C08918=1012.059,211.488,-136.329,-51.249,85.122,-51.521
C08919=1012.057,211.246,-136.302,-51.186,85.113,-51.456
C08920=1012.055,211.003,-136.276,-51.123,85.104,-51.390
C08921=1012.053,210.760,-136.249,-51.059,85.095,-51.325
C08922=1012.051,210.518,-136.223,-50.990,85.086,-51.253
C08923=1012.049,210.275,-136.196,-50.928,85.077,-51.188
C08924=1012.046,210.033,-136.169,-50.865,85.068,-51.124
C08925=1012.044,209.791,-136.143,-50.803,85.060,-51.060
C08926=1012.042,209.548,-136.116,-50.748,85.051,-51.003
C08927=1012.040,209.306,-136.090,-50.679,85.041,-50.932
C08928=1012.037,209.063,-136.063,-50.618,85.032,-50.869
C08929=1012.036,208.821,-136.037,-50.557,85.024,-50.805
C08930=1012.034,208.578,-136.010,-50.495,85.014,-50.742
C08931=1012.032,208.336,-135.984,-50.441,85.007,-50.686
C08932=1012.030,208.093,-135.958,-50.374,84.997,-50.617
C08933=1012.027,207.851,-135.931,-50.314,84.988,-50.555
C08934=1012.025,207.608,-135.905,-50.254,84.979,-50.492
C08935=1012.023,207.365,-135.878,-50.194,84.970,-50.430
C08936=1012.021,207.122,-135.852,-50.134,84.961,-50.369
C08937=1012.020,206.880,-135.826,-50.074,84.951,-50.307
C08938=1012.018,206.636,-135.799,-50.015,84.943,-50.246
C08939=1012.016,206.393,-135.773,-49.956,84.934,-50.185
C08940=1012.014,206.150,-135.746,-49.897,84.924,-50.124
C08941=1012.011,205.906,-135.720,-49.838,84.915,-50.064
C08942=1012.010,205.663,-135.693,-49.780,84.907,-50.003
C08943=1012.008,205.419,-135.667,-49.716,84.897,-49.936
C08944=1012.005,205.175,-135.640,-49.658,84.888,-49.876
C08945=1012.004,204.930,-135.613,-49.600,84.878,-49.817
C08946=1012.002,204.687,-135.587,-49.542,84.870,-49.757
C08947=1011.999,204.443,-135.561,-49.485,84.860,-49.698
C08948=1011.998,204.198,-135.534,-49.422,84.851,-49.632
C08949=1011.996,203.954,-135.508,-49.365,84.841,-49.573
C08950=1011.994,203.710,-135.481,-49.308,84.833,-49.514
C08951=1011.992,203.464,-135.454,-49.251,84.823,-49.456
C08952=1011.987,202.215,-135.317,-47.331,85.025,-47.026
C08953=1011.988,201.996,-135.294,-47.276,85.015,-46.969
C08954=1011.988,201.790,-135.271,-47.227,85.007,-46.919
C08955=1011.988,201.373,-135.226,-47.131,84.989,-46.820
C08956=1011.989,201.157,-135.203,-47.083,84.981,-46.770
C08957=1011.989,200.933,-135.179,-47.029,84.971,-46.714
C08958=1011.989,200.695,-135.153,-46.976,84.962,-46.659
C08959=1011.989,200.439,-135.126,-46.922,84.951,-46.605
C08960=1011.990,200.186,-135.099,-46.863,84.940,-46.544
C08961=1011.989,199.944,-135.073,-46.811,84.930,-46.490
C08962=1011.990,199.712,-135.048,-46.758,84.921,-46.435
C08963=1011.990,199.483,-135.023,-46.705,84.911,-46.381
C08964=1011.990,199.241,-134.997,-46.653,84.902,-46.327
C08965=1011.991,198.850,-134.954,-46.566,84.885,-46.238
C08966=1011.991,198.458,-134.913,-46.486,84.869,-46.156
C08967=1011.992,198.212,-134.886,-46.429,84.859,-46.096
C08968=1011.992,197.976,-134.861,-46.378,84.848,-46.044
C08969=1011.992,197.740,-134.836,-46.327,84.838,-45.991
C08970=1011.992,197.504,-134.810,-46.276,84.829,-45.939
C08971=1011.993,197.268,-134.785,-46.226,84.818,-45.887
C08972=1011.993,197.032,-134.759,-46.175,84.808,-45.835
C08973=1011.993,196.796,-134.734,-46.125,84.799,-45.783
C08974=1011.993,196.560,-134.709,-46.075,84.789,-45.731
C08975=1011.994,196.324,-134.684,-46.031,84.780,-45.686
C08976=1011.994,196.088,-134.658,-45.981,84.770,-45.635
C08977=1011.995,195.852,-134.633,-45.932,84.761,-45.583
C08978=1011.995,195.616,-134.609,-45.883,84.750,-45.533
C08979=1011.995,195.380,-134.583,-45.834,84.740,-45.483
C08980=1011.996,195.144,-134.558,-45.785,84.731,-45.432
C08981=1011.996,194.908,-134.532,-45.742,84.721,-45.388
C08982=1011.996,194.673,-134.507,-45.693,84.711,-45.339
C08983=1011.997,194.437,-134.482,-45.645,84.701,-45.288
C08984=1011.997,194.201,-134.456,-45.602,84.692,-45.245
C08985=1011.998,193.965,-134.431,-45.554,84.682,-45.195
C08986=1011.997,193.729,-134.406,-45.512,84.673,-45.151
C08987=1011.998,193.492,-134.381,-45.464,84.663,-45.102
C08988=1011.999,193.257,-134.356,-45.417,84.653,-45.053
C08989=1011.999,193.021,-134.330,-45.370,84.643,-45.005
C08990=1011.999,192.785,-134.306,-45.323,84.633,-44.956
C08991=1011.999,192.549,-134.280,-45.281,84.624,-44.913
C08992=1012.000,192.313,-134.255,-45.235,84.614,-44.865
C08993=1012.000,192.077,-134.229,-45.188,84.604,-44.817
C08994=1012.000,191.841,-134.205,-45.147,84.595,-44.774
C08995=1012.001,191.605,-134.180,-45.106,84.586,-44.732
C08996=1012.001,191.369,-134.154,-45.060,84.576,-44.685
C08997=1012.002,191.133,-134.129,-45.019,84.567,-44.643
C08998=1012.002,190.898,-134.104,-44.974,84.556,-44.597
C08999=1012.002,190.662,-134.079,-44.928,84.546,-44.549
C09000=1012.003,190.425,-134.054,-44.883,84.537,-44.502
C09001=1012.004,190.189,-134.028,-44.838,84.527,-44.455
C09002=1012.003,189.954,-134.004,-44.798,84.517,-44.415
C09003=1012.004,189.718,-133.978,-44.759,84.507,-44.375
C09004=1012.004,189.482,-133.953,-44.714,84.498,-44.328
C09005=1012.005,189.245,-133.928,-44.674,84.488,-44.288
C09006=1012.006,189.010,-133.903,-44.635,84.480,-44.246
C09007=1012.006,188.774,-133.878,-44.591,84.469,-44.201
C09008=1012.006,188.538,-133.853,-44.547,84.459,-44.155
C09009=1012.007,188.302,-133.828,-44.508,84.450,-44.115
C09010=1012.007,188.066,-133.803,-44.464,84.439,-44.071
C09011=1012.007,187.830,-133.777,-44.421,84.430,-44.026
C09012=1012.008,187.595,-133.753,-44.382,84.420,-43.986
C09013=1012.008,187.359,-133.728,-44.344,84.411,-43.947
C09014=1012.009,187.123,-133.703,-44.306,84.402,-43.907
C09015=1012.010,186.887,-133.677,-44.263,84.392,-43.863
C09016=1012.009,186.651,-133.652,-44.225,84.383,-43.824
C09017=1012.011,186.415,-133.628,-44.187,84.373,-43.785
C09018=1012.011,186.179,-133.603,-44.145,84.363,-43.740
C09019=1012.011,185.943,-133.578,-44.103,84.353,-43.698
C09020=1012.011,185.707,-133.552,-44.065,84.343,-43.659
C09021=1012.013,185.472,-133.528,-44.023,84.334,-43.615
C09022=1012.012,185.236,-133.503,-43.986,84.324,-43.577
C09023=1012.013,185.000,-133.478,-43.949,84.315,-43.539
C09024=1012.014,184.763,-133.453,-43.912,84.306,-43.501
C09025=1012.014,184.528,-133.428,-43.876,84.296,-43.464
C09026=1012.015,184.292,-133.403,-43.839,84.287,-43.426
C09027=1012.015,184.057,-133.377,-43.798,84.277,-43.383
C09028=1012.015,183.820,-133.353,-43.756,84.267,-43.340
C09029=1012.016,183.585,-133.328,-43.721,84.257,-43.304
C09030=1012.017,183.349,-133.303,-43.685,84.248,-43.267
C09031=1012.017,183.113,-133.279,-43.644,84.238,-43.224
C09032=1012.018,182.877,-133.254,-43.608,84.228,-43.188
C09033=1012.018,182.642,-133.228,-43.573,84.219,-43.151
C09034=1012.018,182.405,-133.204,-43.537,84.210,-43.114
C09035=1012.019,182.170,-133.179,-43.502,84.200,-43.078
C09036=1012.020,181.934,-133.153,-43.466,84.191,-43.041
C09037=1012.020,181.698,-133.129,-43.431,84.182,-43.005
C09038=1012.021,181.462,-133.104,-43.391,84.172,-42.963
C09039=1012.021,181.227,-133.079,-43.356,84.162,-42.927
C09040=1012.021,180.990,-133.055,-43.317,84.152,-42.888
C09041=1012.023,180.755,-133.029,-43.283,84.142,-42.852
C09042=1012.023,180.519,-133.005,-43.248,84.133,-42.816
C09043=1012.024,180.283,-132.980,-43.214,84.123,-42.781
C09044=1012.024,180.047,-132.955,-43.179,84.114,-42.745
C09045=1012.024,179.811,-132.931,-43.149,84.106,-42.714
C09046=1012.025,179.576,-132.905,-43.115,84.097,-42.679
C09047=1012.026,179.340,-132.880,-43.077,84.086,-42.640
C09048=1012.026,179.104,-132.856,-43.043,84.077,-42.605
C09049=1012.027,178.868,-132.831,-43.009,84.067,-42.570
C09050=1012.027,178.632,-132.807,-42.971,84.057,-42.530
C09051=1012.028,178.397,-132.782,-42.937,84.048,-42.495
C09052=1012.028,178.161,-132.756,-42.904,84.038,-42.461
C09053=1012.029,177.925,-132.732,-42.875,84.030,-42.432
C09054=1012.030,177.689,-132.707,-42.842,84.020,-42.397
C09055=1012.030,177.454,-132.683,-42.809,84.011,-42.363
C09056=1012.031,177.218,-132.658,-42.776,84.001,-42.329
C09057=1012.032,176.982,-132.633,-42.743,83.992,-42.295
C09058=1012.032,176.746,-132.608,-42.705,83.982,-42.256
C09059=1012.033,176.511,-132.583,-42.673,83.973,-42.222
C09060=1012.033,176.275,-132.559,-42.641,83.962,-42.190
C09061=1012.034,176.040,-132.534,-42.608,83.953,-42.157
C09062=1012.034,175.803,-132.510,-42.576,83.943,-42.123
C09063=1012.035,175.568,-132.485,-42.547,83.936,-42.094
C09064=1012.036,175.331,-132.460,-42.515,83.926,-42.060
C09065=1012.036,175.096,-132.436,-42.483,83.917,-42.027
C09066=1012.037,174.860,-132.410,-42.451,83.907,-41.994
C09067=1012.037,174.625,-132.386,-42.419,83.898,-41.961
C09068=1012.038,174.389,-132.361,-42.388,83.888,-41.930
C09069=1012.038,174.153,-132.337,-42.357,83.878,-41.897
C09070=1012.039,173.917,-132.312,-42.325,83.869,-41.865
C09071=1012.040,173.682,-132.288,-42.294,83.859,-41.832
C09072=1012.040,173.446,-132.262,-42.267,83.850,-41.805
C09073=1012.041,173.210,-132.239,-42.235,83.842,-41.771
C09074=1012.042,172.975,-132.214,-42.204,83.832,-41.739
C09075=1012.043,172.738,-132.189,-42.177,83.824,-41.712
C09076=1012.043,172.504,-132.164,-42.146,83.814,-41.680
C09077=1012.044,172.267,-132.140,-42.115,83.805,-41.648
C09078=1012.044,172.032,-132.115,-42.085,83.794,-41.618
C09079=1012.045,171.796,-132.091,-42.054,83.785,-41.586
C09080=1012.045,171.560,-132.066,-42.024,83.775,-41.554
C09081=1012.047,171.325,-132.041,-41.993,83.766,-41.523
C09082=1012.047,171.090,-132.017,-41.966,83.758,-41.495
C09083=1012.047,170.854,-131.991,-41.936,83.749,-41.463
C09084=1012.048,170.618,-131.968,-41.910,83.740,-41.437
C09085=1012.049,170.383,-131.943,-41.880,83.730,-41.406
C09086=1012.049,170.147,-131.918,-41.850,83.721,-41.375
C09087=1012.050,169.911,-131.894,-41.820,83.711,-41.344
C09088=1012.051,169.676,-131.870,-41.790,83.702,-41.313
C09089=1012.051,169.439,-131.845,-41.765,83.693,-41.287
C09090=1012.052,169.204,-131.820,-41.735,83.683,-41.256
C09091=1012.053,168.969,-131.797,-41.705,83.674,-41.226
C09092=1012.053,168.733,-131.771,-41.680,83.665,-41.200
C09093=1012.054,168.497,-131.747,-41.651,83.656,-41.170
C09094=1012.055,168.262,-131.722,-41.625,83.648,-41.143
C09095=1012.055,168.026,-131.698,-41.600,83.639,-41.117
C09096=1012.056,167.790,-131.673,-41.571,83.629,-41.087
C09097=1012.057,167.555,-131.649,-41.542,83.619,-41.059
C09098=1012.058,167.319,-131.624,-41.513,83.609,-41.029
C09099=1012.058,167.083,-131.600,-41.485,83.600,-40.999
C09100=1012.058,166.848,-131.576,-41.460,83.591,-40.974
C09101=1012.059,166.612,-131.551,-41.430,83.582,-40.942
C09102=1012.060,166.377,-131.527,-41.406,83.573,-40.917
C09103=1012.061,166.142,-131.502,-41.381,83.565,-40.893
C09104=1012.061,165.906,-131.477,-41.353,83.555,-40.863
C09105=1012.062,165.670,-131.453,-41.328,83.547,-40.837
C09106=1012.063,165.434,-131.429,-41.299,83.538,-40.808
C09107=1012.063,165.200,-131.405,-41.275,83.529,-40.783
C09108=1012.064,164.896,-131.373,-41.240,83.517,-40.746
C09109=1012.065,164.578,-131.340,-41.210,83.505,-40.716
C09110=1012.066,164.304,-131.312,-41.179,83.494,-40.684
C09111=1012.067,163.969,-131.277,-41.141,83.481,-40.645
C09112=1012.068,163.749,-131.254,-41.116,83.473,-40.619
C09113=1012.068,163.511,-131.230,-41.092,83.464,-40.595
C09114=1012.069,163.247,-131.202,-41.062,83.453,-40.563
C09115=1012.071,162.954,-131.172,-41.031,83.442,-40.532
C09116=1012.070,162.646,-131.140,-41.001,83.431,-40.501
C09117=1012.072,162.355,-131.110,-40.966,83.419,-40.465
C09118=1012.073,162.048,-131.079,-40.937,83.407,-40.436
C09119=1012.073,161.745,-131.047,-40.903,83.395,-40.400
C09120=1012.075,161.453,-131.017,-40.873,83.384,-40.369
C09121=1012.076,161.175,-130.988,-40.843,83.373,-40.339
C09122=1012.076,160.912,-130.961,-40.816,83.363,-40.311
C09123=1012.077,160.663,-130.935,-40.791,83.353,-40.285
C09124=1012.078,160.422,-130.911,-40.764,83.343,-40.257
C09125=1012.079,160.188,-130.887,-40.741,83.334,-40.234
C09126=1012.080,159.956,-130.865,-40.625,83.289,-40.116
C09127=1012.080,159.723,-130.845,-40.392,83.195,-39.879
C09128=1012.082,159.489,-130.825,-40.163,83.099,-39.646
C09129=1012.083,159.253,-130.805,-39.936,83.004,-39.413
C09130=1012.084,159.017,-130.786,-39.720,82.908,-39.193
C09131=1012.085,158.781,-130.765,-39.510,82.812,-38.979
C09132=1012.086,158.546,-130.745,-39.305,82.716,-38.770
C09133=1012.087,158.311,-130.725,-39.107,82.620,-38.568
C09134=1012.089,158.074,-130.705,-38.914,82.523,-38.371
C09135=1012.090,157.837,-130.685,-38.721,82.427,-38.174
C09136=1012.092,157.599,-130.665,-38.539,82.330,-37.988
C09137=1012.092,157.360,-130.644,-38.358,82.233,-37.803
C09138=1012.093,157.121,-130.624,-38.181,82.135,-37.623
C09139=1012.095,156.882,-130.604,-38.010,82.037,-37.448
C09140=1012.096,156.643,-130.584,-37.842,81.939,-37.277
C09141=1012.097,156.403,-130.563,-37.680,81.841,-37.110
C09142=1012.099,156.163,-130.543,-37.524,81.743,-36.952
C09143=1012.100,155.924,-130.523,-37.368,81.646,-36.792
C09144=1012.101,155.685,-130.503,-37.217,81.548,-36.638
C09145=1012.102,155.446,-130.483,-37.071,81.451,-36.489
C09146=1012.104,155.205,-130.463,-36.927,81.352,-36.342
C09147=1012.105,154.965,-130.442,-36.787,81.253,-36.199
C09148=1012.106,154.725,-130.422,-36.652,81.156,-36.061
C09149=1012.108,154.484,-130.402,-36.518,81.057,-35.925
C09150=1012.109,154.243,-130.381,-36.387,80.959,-35.790
C09151=1012.110,154.002,-130.361,-36.262,80.860,-35.663
C09152=1012.112,153.761,-130.340,-36.136,80.762,-35.534
C09153=1012.113,153.520,-130.320,-36.013,80.664,-35.408
C09154=1012.115,153.277,-130.299,-35.897,80.565,-35.290
C09155=1012.116,153.037,-130.279,-35.780,80.466,-35.170
C09156=1012.118,152.794,-130.259,-35.665,80.368,-35.053
C09157=1012.119,152.553,-130.238,-35.557,80.269,-34.943
C09158=1012.121,152.309,-130.217,-35.447,80.170,-34.831
C09159=1012.122,152.060,-130.196,-35.338,80.068,-34.720
C09160=1012.124,151.805,-130.176,-35.230,79.964,-34.610
C09161=1012.125,151.548,-130.154,-35.122,79.859,-34.500
C09162=1012.126,151.284,-130.131,-35.013,79.751,-34.389
C09163=1012.128,150.992,-130.107,-34.898,79.633,-34.272
C09164=1012.130,150.706,-130.082,-34.786,79.517,-34.158
C09165=1012.132,150.413,-130.057,-34.676,79.397,-34.046
C09166=1012.134,150.117,-130.032,-34.568,79.277,-33.937
C09167=1012.136,149.816,-130.007,-34.461,79.155,-33.828
C09168=1012.137,149.517,-129.981,-34.355,79.033,-33.721
C09169=1012.139,149.217,-129.956,-34.252,78.911,-33.615
C09170=1012.141,148.921,-129.931,-34.154,78.791,-33.517
C09171=1012.143,148.630,-129.907,-34.060,78.672,-33.422
C09172=1012.145,148.344,-129.883,-33.969,78.557,-33.329
C09173=1012.147,148.066,-129.859,-33.883,78.443,-33.242
C09174=1012.149,147.796,-129.837,-33.801,78.334,-33.160
C09175=1012.150,147.535,-129.814,-33.724,78.228,-33.082
C09176=1012.152,147.280,-129.793,-33.650,78.125,-33.007
C09177=1012.153,147.032,-129.772,-33.581,78.024,-32.938
C09178=1012.154,146.788,-129.751,-33.512,77.925,-32.869
C09179=1012.156,146.546,-129.731,-33.445,77.828,-32.801
C09180=1012.158,146.303,-129.710,-33.381,77.730,-32.737
C09181=1012.159,146.061,-129.690,-33.317,77.632,-32.674
C09182=1012.162,145.819,-129.670,-33.254,77.534,-32.610
C09183=1012.163,145.577,-129.649,-33.193,77.436,-32.549
C09184=1012.164,145.335,-129.629,-33.132,77.338,-32.488
C09185=1012.166,145.093,-129.608,-33.073,77.242,-32.430
C09186=1012.168,144.852,-129.588,-33.014,77.144,-32.371
C09187=1012.170,144.611,-129.568,-32.959,77.046,-32.317
C09188=1012.171,144.369,-129.547,-32.903,76.949,-32.262
C09189=1012.172,144.128,-129.527,-32.846,76.852,-32.204
C09190=1012.174,143.887,-129.506,-32.793,76.755,-32.151
C09191=1012.176,143.647,-129.486,-32.741,76.659,-32.101
C09192=1012.178,143.406,-129.466,-32.689,76.562,-32.049
C09193=1012.179,143.166,-129.446,-32.638,76.465,-31.999
C09194=1012.181,142.925,-129.425,-32.588,76.370,-31.950
C09195=1012.183,142.686,-129.404,-32.539,76.272,-31.902
C09196=1012.185,142.446,-129.385,-32.490,76.176,-31.855
C09197=1012.186,142.207,-129.365,-32.443,76.081,-31.808
C09198=1012.188,141.968,-129.344,-32.396,75.985,-31.763
C09199=1012.190,141.729,-129.324,-32.351,75.889,-31.718
C09200=1012.192,141.484,-129.304,-32.305,75.791,-31.675
C09201=1012.193,141.273,-129.286,-32.265,75.707,-31.635
C09202=1012.195,141.017,-129.264,-32.219,75.605,-31.591
C09203=1012.196,140.845,-129.249,-32.188,75.536,-31.561
C09204=1012.199,140.472,-129.219,-32.123,75.387,-31.499
C09205=1012.201,140.197,-129.195,-32.074,75.279,-31.452
C09206=1012.203,139.902,-129.170,-32.023,75.160,-31.403
C09207=1012.206,139.593,-129.144,-31.973,75.037,-31.355
C09208=1012.208,139.280,-129.118,-31.922,74.913,-31.307
C09209=1012.211,138.972,-129.092,-31.873,74.791,-31.261
C09210=1012.213,138.678,-129.067,-31.826,74.674,-31.216
C09211=1012.214,138.404,-129.044,-31.784,74.565,-31.177
C09212=1012.216,138.152,-129.022,-31.747,74.466,-31.143
C09213=1012.220,137.732,-128.987,-31.684,74.299,-31.084
C09214=1012.223,137.348,-128.955,-31.630,74.147,-31.034
C09215=1012.226,136.931,-128.919,-31.571,73.983,-30.980
C09216=1012.228,136.548,-128.887,-31.518,73.831,-30.932
C09217=1012.232,136.162,-128.854,-31.466,73.679,-30.883
C09218=1012.235,135.743,-128.819,-31.413,73.514,-30.837
C09219=1012.237,135.518,-128.801,-31.383,73.426,-30.810
C09220=1012.239,135.285,-128.781,-31.354,73.335,-30.784
C09221=1012.241,134.999,-128.756,-31.318,73.222,-30.752
C09222=1012.243,134.704,-128.731,-31.282,73.106,-30.720
C09223=1012.245,134.464,-128.711,-31.254,73.013,-30.696
C09224=1012.247,134.229,-128.691,-31.225,72.921,-30.670
C09225=1012.249,133.993,-128.672,-31.198,72.830,-30.647
C09226=1012.251,133.758,-128.652,-31.171,72.738,-30.623
C09227=1012.253,133.523,-128.632,-31.145,72.646,-30.602
C09228=1012.254,133.288,-128.612,-31.118,72.555,-30.578
C09229=1012.257,133.053,-128.592,-31.092,72.464,-30.556
C09230=1012.258,132.817,-128.573,-31.067,72.372,-30.535
C09231=1012.260,132.582,-128.553,-31.042,72.280,-30.513
C09232=1012.262,132.347,-128.533,-31.017,72.189,-30.493
C09233=1012.264,132.112,-128.513,-30.992,72.099,-30.472
C09234=1012.266,131.876,-128.493,-30.968,72.007,-30.452
C09235=1012.268,131.641,-128.473,-30.944,71.917,-30.432
C09236=1012.270,131.406,-128.453,-30.921,71.826,-30.414
C09237=1012.271,131.171,-128.433,-30.897,71.735,-30.393
C09238=1012.274,130.936,-128.413,-30.874,71.644,-30.376
C09239=1012.275,130.701,-128.393,-30.851,71.554,-30.358
C09240=1012.278,130.466,-128.373,-30.829,71.463,-30.340
C09241=1012.279,130.230,-128.353,-30.807,71.373,-30.322
C09242=1012.282,129.995,-128.333,-30.785,71.283,-30.306
C09243=1012.283,129.760,-128.314,-30.764,71.193,-30.289
C09244=1012.286,129.525,-128.294,-30.742,71.103,-30.272
C09245=1012.287,129.289,-128.274,-30.722,71.013,-30.257
C09246=1012.290,129.054,-128.254,-30.701,70.923,-30.242
C09247=1012.291,128.819,-128.234,-30.680,70.833,-30.226
C09248=1012.293,128.584,-128.214,-30.660,70.744,-30.210
C09249=1012.295,128.349,-128.195,-30.640,70.654,-30.196
C09250=1012.297,128.114,-128.175,-30.621,70.565,-30.182
C09251=1012.299,127.878,-128.155,-30.601,70.476,-30.167
C09252=1012.301,127.643,-128.135,-30.582,70.387,-30.153
C09253=1012.303,127.408,-128.115,-30.563,70.297,-30.140
C09254=1012.305,127.173,-128.095,-30.544,70.209,-30.127
C09255=1012.307,126.937,-128.075,-30.525,70.120,-30.113
C09256=1012.309,126.702,-128.056,-30.508,70.030,-30.103
C09257=1012.312,126.467,-128.036,-30.489,69.941,-30.089
C09258=1012.313,126.232,-128.016,-30.472,69.853,-30.078
C09259=1012.316,125.997,-127.996,-30.454,69.765,-30.066
C09260=1012.317,125.762,-127.975,-30.437,69.676,-30.055
C09261=1012.319,125.527,-127.956,-30.420,69.588,-30.044
C09262=1012.321,125.292,-127.935,-30.402,69.500,-30.031
C09263=1012.323,125.057,-127.916,-30.386,69.412,-30.021
C09264=1012.326,124.822,-127.896,-30.369,69.324,-30.011
C09265=1012.327,124.587,-127.877,-30.353,69.237,-30.000
C09266=1012.330,124.352,-127.857,-30.336,69.148,-29.991
C09267=1012.332,124.116,-127.836,-30.320,69.061,-29.981
C09268=1012.334,123.881,-127.817,-30.304,68.973,-29.971
C09269=1012.336,123.645,-127.797,-30.289,68.886,-29.962
C09270=1012.338,123.411,-127.777,-30.273,68.799,-29.953
C09271=1012.340,123.176,-127.757,-30.258,68.711,-29.945
C09272=1012.342,122.940,-127.737,-30.243,68.624,-29.937
C09273=1012.344,122.705,-127.718,-30.228,68.537,-29.928
C09274=1012.346,122.470,-127.697,-30.213,68.450,-29.920
C09275=1012.348,122.235,-127.678,-30.198,68.363,-29.911
C09276=1012.350,122.001,-127.657,-30.184,68.277,-29.905
C09277=1012.353,121.692,-127.631,-30.165,68.164,-29.895
C09278=1012.357,121.295,-127.598,-30.141,68.018,-29.883
C09279=1012.359,121.059,-127.577,-30.128,67.931,-29.877
C09280=1012.361,120.825,-127.558,-30.114,67.844,-29.870
C09281=1012.363,120.589,-127.538,-30.100,67.754,-29.864
C09282=1012.365,120.354,-127.518,-30.085,67.660,-29.856
C09283=1012.368,120.119,-127.499,-30.070,67.567,-29.850
C09284=1012.369,119.884,-127.480,-30.056,67.472,-29.845
C09285=1012.372,119.649,-127.460,-30.042,67.379,-29.839
C09286=1012.374,119.414,-127.441,-30.027,67.286,-29.832
C09287=1012.376,119.179,-127.420,-30.014,67.193,-29.827
C09288=1012.378,118.943,-127.402,-30.000,67.099,-29.822
C09289=1012.381,118.708,-127.382,-29.987,67.006,-29.817
C09290=1012.383,118.473,-127.362,-29.973,66.912,-29.811
C09291=1012.385,118.239,-127.342,-29.960,66.820,-29.807
C09292=1012.388,118.003,-127.323,-29.947,66.727,-29.803
C09293=1012.390,117.768,-127.304,-29.933,66.635,-29.797
C09294=1012.392,117.533,-127.284,-29.920,66.541,-29.793
C09295=1012.394,117.298,-127.264,-29.908,66.449,-29.791
C09296=1012.397,117.063,-127.244,-29.895,66.357,-29.786
C09297=1012.399,116.828,-127.226,-29.883,66.264,-29.783
C09298=1012.401,116.593,-127.206,-29.870,66.172,-29.780
C09299=1012.404,116.357,-127.185,-29.858,66.080,-29.778
C09300=1012.405,116.122,-127.166,-29.845,65.987,-29.774
C09301=1012.408,115.887,-127.147,-29.834,65.897,-29.772
C09302=1012.410,115.652,-127.127,-29.822,65.804,-29.770
C09303=1012.413,115.417,-127.108,-29.810,65.712,-29.767
C09304=1012.415,115.182,-127.088,-29.799,65.620,-29.765
C09305=1012.417,114.947,-127.068,-29.787,65.529,-29.764
C09306=1012.420,114.711,-127.049,-29.776,65.438,-29.761
C09307=1012.422,114.476,-127.029,-29.765,65.347,-29.760
C09308=1012.424,114.241,-127.009,-29.754,65.256,-29.760
C09309=1012.427,114.006,-126.989,-29.742,65.165,-29.756
C09310=1012.429,113.772,-126.970,-29.731,65.073,-29.756
C09311=1012.432,113.536,-126.951,-29.720,64.982,-29.755
C09312=1012.434,113.301,-126.932,-29.709,64.892,-29.754
C09313=1012.436,113.066,-126.911,-29.699,64.802,-29.755
C09314=1012.438,112.831,-126.891,-29.688,64.711,-29.753
C09315=1012.440,112.596,-126.872,-29.678,64.620,-29.754
C09316=1012.443,112.360,-126.853,-29.667,64.531,-29.754
C09317=1012.446,112.125,-126.833,-29.657,64.440,-29.755
C09318=1012.447,111.891,-126.813,-29.647,64.350,-29.754
C09319=1012.450,111.656,-126.794,-29.637,64.260,-29.755
C09320=1012.451,111.420,-126.774,-29.627,64.171,-29.755
C09321=1012.454,111.185,-126.755,-29.617,64.081,-29.756
C09322=1012.457,110.950,-126.735,-29.607,63.991,-29.757
C09323=1012.459,110.715,-126.715,-29.597,63.902,-29.758
C09324=1012.461,110.480,-126.695,-29.588,63.813,-29.760
C09325=1012.464,110.245,-126.675,-29.578,63.723,-29.761
C09326=1012.466,110.010,-126.657,-29.569,63.634,-29.763
C09327=1012.469,109.775,-126.637,-29.559,63.545,-29.763
C09328=1012.471,109.539,-126.617,-29.550,63.456,-29.766
C09329=1012.473,109.304,-126.597,-29.541,63.367,-29.769
C09330=1012.475,109.069,-126.577,-29.531,63.279,-29.770
C09331=1012.478,108.834,-126.557,-29.522,63.190,-29.773
C09332=1012.480,108.599,-126.539,-29.513,63.102,-29.775
C09333=1012.483,108.364,-126.519,-29.504,63.014,-29.777
C09334=1012.486,108.129,-126.499,-29.495,62.926,-29.781
C09335=1012.487,107.894,-126.479,-29.486,62.837,-29.783
C09336=1012.489,107.658,-126.459,-29.478,62.750,-29.786
C09337=1012.492,107.423,-126.440,-29.469,62.663,-29.789
C09338=1012.495,107.188,-126.420,-29.460,62.574,-29.792
C09339=1012.497,106.953,-126.401,-29.452,62.487,-29.795
C09340=1012.499,106.718,-126.381,-29.443,62.399,-29.799
C09341=1012.503,106.403,-126.354,-29.432,62.282,-29.805
C09342=1012.506,106.012,-126.322,-29.418,62.138,-29.811
C09343=1012.509,105.777,-126.302,-29.410,62.051,-29.814
C09344=1012.511,105.542,-126.283,-29.402,61.964,-29.819
C09345=1012.513,105.307,-126.263,-29.394,61.877,-29.823
C09346=1012.516,105.072,-126.243,-29.386,61.791,-29.827
C09347=1012.519,104.837,-126.223,-29.378,61.704,-29.832
C09348=1012.521,104.602,-126.204,-29.370,61.618,-29.836
C09349=1012.524,104.367,-126.184,-29.362,61.532,-29.841
C09350=1012.526,104.131,-126.164,-29.354,61.445,-29.846
C09351=1012.528,103.896,-126.144,-29.346,61.359,-29.851
C09352=1012.530,103.662,-126.125,-29.339,61.274,-29.856
C09353=1012.533,103.426,-126.105,-29.331,61.188,-29.861
C09354=1012.536,103.191,-126.085,-29.323,61.103,-29.866
C09355=1012.538,102.956,-126.065,-29.316,61.017,-29.872
C09356=1012.540,102.721,-126.046,-29.308,60.932,-29.878
C09357=1012.542,102.486,-126.026,-29.301,60.846,-29.883
C09358=1012.545,102.251,-126.006,-29.294,60.762,-29.890
C09359=1012.548,102.015,-125.987,-29.286,60.677,-29.894
C09360=1012.550,101.780,-125.967,-29.279,60.592,-29.901
C09361=1012.552,101.545,-125.947,-29.271,60.507,-29.905
C09362=1012.555,101.310,-125.927,-29.264,60.423,-29.913
C09363=1012.557,101.075,-125.907,-29.257,60.339,-29.919
C09364=1012.559,100.840,-125.888,-29.250,60.254,-29.925
C09365=1012.562,100.604,-125.869,-29.243,60.170,-29.931
C09366=1012.564,100.369,-125.849,-29.235,60.086,-29.937
C09367=1012.567,100.134,-125.829,-29.228,60.003,-29.944
C09368=1012.569,99.900,-125.809,-29.222,59.920,-29.951
C09369=1012.571,99.664,-125.789,-29.214,59.836,-29.957
C09370=1012.573,99.429,-125.769,-29.208,59.753,-29.965
C09371=1012.576,99.193,-125.750,-29.201,59.669,-29.971
C09372=1012.579,98.958,-125.730,-29.194,59.586,-29.979
C09373=1012.581,98.724,-125.711,-29.187,59.503,-29.987
C09374=1012.583,98.488,-125.690,-29.181,59.421,-29.993
C09375=1012.586,98.253,-125.670,-29.174,59.338,-30.001
C09376=1012.588,98.018,-125.650,-29.167,59.257,-30.008
C09377=1012.591,97.782,-125.631,-29.161,59.174,-30.016
C09378=1012.593,97.548,-125.612,-29.154,59.092,-30.024
C09379=1012.595,97.312,-125.591,-29.147,59.010,-30.030
C09380=1012.598,97.077,-125.572,-29.141,58.928,-30.040
C09381=1012.600,96.842,-125.552,-29.135,58.847,-30.047
C09382=1012.603,96.607,-125.532,-29.128,58.765,-30.055
C09383=1012.606,96.371,-125.512,-29.122,58.684,-30.063
C09384=1012.607,96.136,-125.493,-29.115,58.602,-30.071
C09385=1012.610,95.901,-125.473,-29.109,58.522,-30.080
C09386=1012.612,95.666,-125.453,-29.103,58.441,-30.087
C09387=1012.615,95.431,-125.433,-29.097,58.360,-30.096
C09388=1012.617,95.195,-125.413,-29.090,58.280,-30.105
C09389=1012.619,94.960,-125.394,-29.084,58.200,-30.112
C09390=1012.622,94.725,-125.374,-29.078,58.119,-30.122
C09391=1012.624,94.490,-125.354,-29.072,58.039,-30.130
C09392=1012.627,94.254,-125.334,-29.066,57.959,-30.139
C09393=1012.629,94.019,-125.314,-29.060,57.880,-30.148
C09394=1012.632,93.784,-125.294,-29.053,57.800,-30.156
C09395=1012.635,93.549,-125.275,-29.047,57.721,-30.165
C09396=1012.636,93.313,-125.255,-29.041,57.642,-30.174
C09397=1012.639,93.078,-125.235,-29.035,57.563,-30.183
C09398=1012.641,92.843,-125.215,-29.030,57.484,-30.193
C09399=1012.644,92.608,-125.195,-29.024,57.404,-30.202
C09400=1012.646,92.373,-125.175,-29.018,57.325,-30.211
C09401=1012.649,92.137,-125.156,-29.012,57.246,-30.221
C09402=1012.651,91.902,-125.136,-29.006,57.169,-30.229
C09403=1012.653,91.667,-125.116,-29.000,57.090,-30.240
C09404=1012.655,91.432,-125.096,-28.994,57.013,-30.249
C09405=1012.658,91.197,-125.076,-28.988,56.934,-30.259
C09406=1012.660,90.960,-125.056,-28.983,56.857,-30.268
C09407=1012.663,90.701,-125.034,-28.977,56.771,-30.280
C09408=1012.666,90.382,-125.008,-28.969,56.666,-30.292
C09409=1012.670,90.049,-124.979,-28.961,56.557,-30.306
C09410=1012.673,89.669,-124.947,-28.952,56.432,-30.323
C09411=1012.677,89.296,-124.916,-28.943,56.311,-30.340
C09412=1012.680,89.066,-124.896,-28.937,56.236,-30.350
C09413=1012.682,88.840,-124.877,-28.932,56.163,-30.359
C09414=1012.684,88.615,-124.858,-28.927,56.090,-30.369
C09415=1012.686,88.390,-124.839,-28.921,56.018,-30.379
C09416=1012.689,88.168,-124.820,-28.916,55.946,-30.388
C09417=1012.691,87.942,-124.802,-28.911,55.873,-30.398
C09418=1012.693,87.716,-124.782,-28.905,55.801,-30.409
C09419=1012.695,87.485,-124.763,-28.900,55.726,-30.420
C09420=1012.699,87.251,-124.743,-28.895,55.652,-30.431
C09421=1012.701,87.015,-124.723,-28.889,55.577,-30.441
C09422=1012.703,86.777,-124.702,-28.884,55.501,-30.451
C09423=1012.706,86.539,-124.683,-28.878,55.425,-30.462
C09424=1012.707,86.299,-124.662,-28.873,55.350,-30.473
C09425=1012.710,86.059,-124.642,-28.867,55.274,-30.485
C09426=1012.712,85.820,-124.621,-28.862,55.199,-30.495
C09427=1012.715,85.580,-124.601,-28.857,55.123,-30.507
C09428=1012.717,85.339,-124.581,-28.851,55.048,-30.518
C09429=1012.720,85.098,-124.561,-28.846,54.972,-30.530
C09430=1012.723,84.857,-124.541,-28.840,54.897,-30.541
C09431=1012.724,84.614,-124.520,-28.835,54.821,-30.553
C09432=1012.727,84.372,-124.500,-28.829,54.745,-30.564
C09433=1012.729,84.129,-124.478,-28.824,54.670,-30.575
C09434=1012.732,83.885,-124.458,-28.819,54.594,-30.588
C09435=1012.734,83.641,-124.437,-28.813,54.520,-30.599
C09436=1012.736,83.397,-124.416,-28.808,54.444,-30.612
C09437=1012.740,83.152,-124.396,-28.802,54.368,-30.623
C09438=1012.742,82.907,-124.375,-28.797,54.293,-30.634
C09439=1012.744,82.661,-124.354,-28.792,54.218,-30.648
C09440=1012.747,82.415,-124.333,-28.786,54.143,-30.659
C09441=1012.749,82.169,-124.312,-28.781,54.068,-30.671
C09442=1012.752,81.923,-124.292,-28.776,53.993,-30.685
C09443=1012.754,81.676,-124.271,-28.770,53.918,-30.696
C09444=1012.756,81.429,-124.250,-28.765,53.843,-30.708
C09445=1012.759,81.186,-124.230,-28.760,53.771,-30.720
C09446=1012.761,80.957,-124.210,-28.755,53.701,-30.733
C09447=1012.762,80.741,-124.191,-28.750,53.637,-30.743
C09448=1012.765,80.523,-124.173,-28.746,53.571,-30.755
C09449=1012.768,80.294,-124.154,-28.741,53.503,-30.767
C09450=1012.770,80.052,-124.133,-28.735,53.430,-30.779
C09451=1012.773,79.805,-124.112,-28.730,53.357,-30.791
C09452=1012.775,79.560,-124.092,-28.725,53.285,-30.804
C09453=1012.777,79.319,-124.071,-28.720,53.214,-30.816
C09454=1012.779,79.079,-124.050,-28.715,53.143,-30.828
C09455=1012.781,78.842,-124.030,-28.710,53.073,-30.841
C09456=1012.784,78.607,-124.010,-28.705,53.003,-30.854
C09457=1012.786,78.375,-123.990,-28.700,52.937,-30.865
C09458=1012.789,78.144,-123.971,-28.695,52.869,-30.877
C09459=1012.791,77.916,-123.952,-28.691,52.803,-30.889
C09460=1012.793,77.689,-123.932,-28.686,52.736,-30.901
C09461=1012.795,77.461,-123.913,-28.681,52.670,-30.913
C09462=1012.797,77.234,-123.893,-28.676,52.604,-30.925
C09463=1012.799,77.005,-123.875,-28.671,52.538,-30.937
C09464=1012.802,76.775,-123.855,-28.667,52.471,-30.950
C09465=1012.804,76.542,-123.835,-28.662,52.405,-30.962
C09466=1012.807,76.307,-123.816,-28.657,52.337,-30.975
C09467=1012.808,76.069,-123.795,-28.652,52.269,-30.988
C09468=1012.811,75.827,-123.775,-28.647,52.201,-31.000
C09469=1012.813,75.584,-123.753,-28.642,52.131,-31.013
C09470=1012.816,75.339,-123.733,-28.637,52.061,-31.027
C09471=1012.818,75.091,-123.712,-28.632,51.991,-31.040
C09472=1012.820,74.842,-123.691,-28.627,51.922,-31.053
C09473=1012.823,74.583,-123.669,-28.622,51.848,-31.068
C09474=1012.825,74.310,-123.646,-28.616,51.772,-31.082
C09475=1012.828,74.043,-123.623,-28.611,51.698,-31.096
C09476=1012.830,73.792,-123.601,-28.606,51.627,-31.111
C09477=1012.833,73.546,-123.580,-28.601,51.559,-31.124
C09478=1012.835,73.301,-123.560,-28.596,51.491,-31.137
C09479=1012.837,73.056,-123.538,-28.591,51.423,-31.150
C09480=1012.839,72.812,-123.518,-28.586,51.356,-31.164
C09481=1012.842,72.568,-123.497,-28.581,51.288,-31.178
C09482=1012.844,72.326,-123.477,-28.576,51.222,-31.190
C09483=1012.847,72.083,-123.456,-28.572,51.156,-31.204
C09484=1012.849,71.842,-123.436,-28.567,51.089,-31.218
C09485=1012.851,71.601,-123.415,-28.562,51.024,-31.231
C09486=1012.853,71.359,-123.395,-28.557,50.959,-31.245
C09487=1012.855,71.118,-123.374,-28.552,50.894,-31.257
C09488=1012.857,70.877,-123.353,-28.548,50.829,-31.271
C09489=1012.860,70.636,-123.333,-28.543,50.764,-31.285
C09490=1012.862,70.395,-123.313,-28.538,50.699,-31.299
C09491=1012.865,70.067,-123.284,-28.532,50.612,-31.317
C09492=1012.869,69.672,-123.250,-28.524,50.506,-31.338
C09493=1012.871,69.431,-123.230,-28.519,50.442,-31.352
C09494=1012.873,69.188,-123.210,-28.514,50.378,-31.366
C09495=1012.876,68.942,-123.189,-28.510,50.314,-31.379
C09496=1012.878,68.694,-123.167,-28.505,50.248,-31.393
C09497=1012.880,68.445,-123.146,-28.500,50.183,-31.407
C09498=1012.883,68.195,-123.125,-28.495,50.118,-31.421
C09499=1012.884,67.951,-123.104,-28.490,50.055,-31.435
C09500=1012.887,67.709,-123.083,-28.486,49.992,-31.449
C09501=1012.889,67.470,-123.063,-28.481,49.930,-31.462
C09502=1012.891,67.233,-123.043,-28.476,49.868,-31.475
C09503=1012.894,66.995,-123.022,-28.472,49.807,-31.489
C09504=1012.895,66.758,-123.002,-28.467,49.747,-31.503
C09505=1012.898,66.523,-122.983,-28.463,49.686,-31.516
C09506=1012.900,66.310,-122.964,-28.458,49.632,-31.528
C09507=1012.903,65.917,-122.931,-28.451,49.532,-31.551
C09508=1012.905,65.685,-122.911,-28.447,49.473,-31.564
C09509=1012.907,65.442,-122.890,-28.442,49.412,-31.578
C09510=1012.910,65.190,-122.868,-28.437,49.348,-31.592
C09511=1012.912,64.929,-122.846,-28.432,49.283,-31.606
C09512=1012.914,64.664,-122.823,-28.427,49.217,-31.622
C09513=1012.916,64.393,-122.801,-28.422,49.149,-31.637
C09514=1012.919,64.126,-122.778,-28.417,49.083,-31.653
C09515=1012.921,63.874,-122.757,-28.412,49.020,-31.667
C09516=1012.923,63.636,-122.736,-28.407,48.961,-31.681
C09517=1012.925,63.385,-122.714,-28.403,48.900,-31.695
C09518=1012.928,63.102,-122.691,-28.397,48.831,-31.711
C09519=1012.930,62.807,-122.665,-28.392,48.759,-31.728
C09520=1012.933,62.532,-122.642,-28.387,48.692,-31.744
C09521=1012.936,62.244,-122.618,-28.381,48.622,-31.761
C09522=1012.938,61.968,-122.594,-28.376,48.555,-31.777
C09523=1012.940,61.732,-122.574,-28.372,48.499,-31.791
C09524=1012.942,61.496,-122.553,-28.367,48.442,-31.804
C09525=1012.944,61.261,-122.533,-28.363,48.387,-31.817
C09526=1012.946,61.025,-122.513,-28.358,48.330,-31.831
C09527=1012.948,60.789,-122.493,-28.354,48.274,-31.845
C09528=1012.949,60.554,-122.473,-28.350,48.219,-31.857
C09529=1012.952,60.317,-122.453,-28.345,48.162,-31.872
C09530=1012.954,60.082,-122.433,-28.341,48.107,-31.884
C09531=1012.956,59.847,-122.413,-28.337,48.052,-31.898
C09532=1012.958,59.611,-122.393,-28.332,47.998,-31.911
C09533=1012.960,59.375,-122.372,-28.328,47.942,-31.926
C09534=1012.962,59.140,-122.353,-28.324,47.887,-31.939
C09535=1012.964,58.904,-122.332,-28.319,47.833,-31.953
C09536=1012.966,58.669,-122.312,-28.315,47.780,-31.966
C09537=1012.968,58.433,-122.292,-28.311,47.725,-31.979
C09538=1012.970,58.197,-122.271,-28.306,47.670,-31.993
C09539=1012.972,57.961,-122.251,-28.302,47.618,-32.006
C09540=1012.973,57.726,-122.231,-28.298,47.564,-32.020
C09541=1012.975,57.490,-122.211,-28.293,47.511,-32.033
C09542=1012.977,57.254,-122.192,-28.289,47.457,-32.048
C09543=1012.979,57.018,-122.171,-28.285,47.404,-32.061
C09544=1012.981,56.783,-122.151,-28.281,47.351,-32.074
C09545=1012.983,56.548,-122.132,-28.276,47.299,-32.087
C09546=1012.985,56.312,-122.111,-28.272,47.247,-32.100
C09547=1012.987,56.076,-122.091,-28.268,47.194,-32.114
C09548=1012.989,55.841,-122.071,-28.264,47.142,-32.128
C09549=1012.991,55.605,-122.050,-28.259,47.090,-32.142
C09550=1012.993,55.370,-122.031,-28.255,47.038,-32.156
C09551=1012.995,55.134,-122.010,-28.251,46.987,-32.168
C09552=1012.997,54.898,-121.990,-28.247,46.935,-32.182
C09553=1012.999,54.662,-121.970,-28.243,46.885,-32.195
C09554=1013.000,54.427,-121.950,-28.238,46.834,-32.208
C09555=1013.002,54.191,-121.930,-28.234,46.783,-32.223
C09556=1013.004,53.956,-121.909,-28.230,46.733,-32.236
C09557=1013.006,53.720,-121.889,-28.226,46.682,-32.249
C09558=1013.007,53.485,-121.869,-28.222,46.632,-32.263
C09559=1013.009,53.249,-121.849,-28.218,46.582,-32.276
C09560=1013.011,53.013,-121.829,-28.213,46.533,-32.288
C09561=1013.013,52.777,-121.808,-28.209,46.483,-32.302
C09562=1013.015,52.542,-121.789,-28.205,46.433,-32.316
C09563=1013.017,52.306,-121.768,-28.201,46.384,-32.328
C09564=1013.019,52.071,-121.748,-28.197,46.335,-32.342
C09565=1013.021,51.835,-121.728,-28.193,46.287,-32.356
C09566=1013.022,51.600,-121.708,-28.189,46.238,-32.368
C09567=1013.024,51.364,-121.688,-28.185,46.190,-32.382
C09568=1013.026,51.128,-121.668,-28.181,46.142,-32.394
C09569=1013.027,50.893,-121.648,-28.177,46.094,-32.408
C09570=1013.030,50.657,-121.628,-28.172,46.046,-32.421
C09571=1013.032,50.422,-121.608,-28.168,45.998,-32.435
C09572=1013.033,50.187,-121.588,-28.164,45.950,-32.448
C09573=1013.035,49.951,-121.568,-28.160,45.904,-32.461
C09574=1013.037,49.715,-121.547,-28.156,45.856,-32.474
C09575=1013.039,49.480,-121.528,-28.152,45.810,-32.487
C09576=1013.041,49.244,-121.507,-28.148,45.763,-32.501
C09577=1013.043,49.008,-121.487,-28.144,45.716,-32.513
C09578=1013.044,48.774,-121.466,-28.140,45.670,-32.526
C09579=1013.046,48.538,-121.446,-28.136,45.625,-32.539
C09580=1013.047,48.302,-121.426,-28.132,45.578,-32.552
C09581=1013.049,48.067,-121.406,-28.129,45.533,-32.566
C09582=1013.051,47.831,-121.386,-28.125,45.487,-32.579
C09583=1013.052,47.596,-121.366,-28.121,45.442,-32.592
C09584=1013.054,47.360,-121.346,-28.117,45.397,-32.604
C09585=1013.056,47.125,-121.326,-28.113,45.352,-32.618
C09586=1013.058,46.889,-121.306,-28.109,45.307,-32.630
C09587=1013.060,46.653,-121.286,-28.105,45.262,-32.643
C09588=1013.061,46.418,-121.266,-28.101,45.218,-32.656
C09589=1013.063,46.183,-121.245,-28.097,45.174,-32.669
C09590=1013.064,45.947,-121.225,-28.093,45.130,-32.681
C09591=1013.066,45.712,-121.205,-28.090,45.087,-32.694
C09592=1013.067,45.476,-121.185,-28.086,45.043,-32.707
C09593=1013.069,45.240,-121.165,-28.082,44.999,-32.720
C09594=1013.071,45.005,-121.144,-28.078,44.956,-32.733
C09595=1013.073,44.769,-121.125,-28.074,44.913,-32.747
C09596=1013.074,44.534,-121.104,-28.070,44.870,-32.758
C09597=1013.076,44.299,-121.084,-28.067,44.827,-32.772
C09598=1013.078,44.063,-121.064,-28.063,44.785,-32.784
C09599=1013.079,43.838,-121.045,-28.059,44.745,-32.795
C09600=1013.081,43.612,-121.026,-28.056,44.704,-32.808
C09601=1013.083,43.357,-121.004,-28.052,44.659,-32.822
C09602=1013.085,43.122,-120.983,-28.048,44.617,-32.834
C09603=1013.086,42.887,-120.964,-28.044,44.576,-32.847
C09604=1013.088,42.651,-120.943,-28.040,44.535,-32.859
C09605=1013.089,42.416,-120.924,-28.037,44.494,-32.872
C09606=1013.091,42.180,-120.904,-28.033,44.452,-32.884
C09607=1013.092,41.945,-120.883,-28.029,44.413,-32.896
C09608=1013.094,41.710,-120.863,-28.026,44.372,-32.909
C09609=1013.096,41.474,-120.843,-28.022,44.331,-32.921
C09610=1013.097,41.239,-120.823,-28.018,44.291,-32.935
C09611=1013.099,41.003,-120.803,-28.015,44.251,-32.946
C09612=1013.100,40.768,-120.782,-28.011,44.211,-32.959
C09613=1013.102,40.533,-120.762,-28.007,44.172,-32.971
C09614=1013.103,40.297,-120.742,-28.004,44.133,-32.983
C09615=1013.104,40.062,-120.723,-28.000,44.093,-32.996
C09616=1013.106,39.827,-120.702,-27.996,44.055,-33.006
C09617=1013.107,39.591,-120.682,-27.993,44.016,-33.019
C09618=1013.109,39.356,-120.662,-27.990,43.977,-33.032
C09619=1013.111,39.120,-120.642,-27.986,43.939,-33.043
C09620=1013.112,38.885,-120.621,-27.982,43.901,-33.055
C09621=1013.114,38.650,-120.601,-27.979,43.862,-33.068
C09622=1013.115,38.414,-120.581,-27.975,43.825,-33.080
C09623=1013.116,38.179,-120.562,-27.972,43.788,-33.092
C09624=1013.118,37.944,-120.541,-27.968,43.750,-33.104
C09625=1013.119,37.709,-120.521,-27.965,43.713,-33.116
C09626=1013.121,37.473,-120.501,-27.961,43.675,-33.128
C09627=1013.123,37.237,-120.481,-27.958,43.639,-33.139
C09628=1013.124,37.003,-120.461,-27.954,43.602,-33.151
C09629=1013.125,36.767,-120.441,-27.951,43.566,-33.163
C09630=1013.127,36.532,-120.421,-27.948,43.530,-33.174
C09631=1013.129,36.297,-120.400,-27.944,43.494,-33.186
C09632=1013.130,36.062,-120.381,-27.941,43.457,-33.198
C09633=1013.131,35.827,-120.361,-27.937,43.422,-33.210
C09634=1013.133,35.591,-120.341,-27.934,43.387,-33.221
C09635=1013.134,35.356,-120.320,-27.931,43.352,-33.233
C09636=1013.135,35.121,-120.301,-27.927,43.317,-33.245
C09637=1013.137,34.885,-120.280,-27.924,43.281,-33.256
C09638=1013.138,34.650,-120.260,-27.921,43.247,-33.267
C09639=1013.140,34.415,-120.240,-27.918,43.213,-33.279
C09640=1013.141,34.180,-120.220,-27.914,43.177,-33.291
C09641=1013.143,33.944,-120.199,-27.911,43.144,-33.302
C09642=1013.144,33.709,-120.180,-27.908,43.110,-33.313
C09643=1013.145,33.474,-120.160,-27.904,43.077,-33.323
C09644=1013.146,33.239,-120.140,-27.901,43.042,-33.336
C09645=1013.148,33.003,-120.120,-27.898,43.010,-33.347
C09646=1013.150,32.768,-120.100,-27.895,42.976,-33.358
C09647=1013.151,32.533,-120.079,-27.892,42.944,-33.369
C09648=1013.152,32.298,-120.059,-27.888,42.911,-33.380
C09649=1013.153,32.062,-120.040,-27.885,42.878,-33.391
C09650=1013.154,31.827,-120.019,-27.882,42.846,-33.403
C09651=1013.156,31.592,-119.999,-27.879,42.814,-33.413
C09652=1013.157,31.356,-119.979,-27.876,42.783,-33.424
C09653=1013.158,31.122,-119.959,-27.873,42.750,-33.436
C09654=1013.160,30.886,-119.939,-27.870,42.719,-33.447
C09655=1013.161,30.651,-119.919,-27.867,42.687,-33.457
C09656=1013.162,30.416,-119.899,-27.864,42.656,-33.468
C09657=1013.163,30.181,-119.879,-27.861,42.625,-33.479
C09658=1013.165,29.946,-119.858,-27.858,42.594,-33.490
C09659=1013.166,29.710,-119.839,-27.855,42.564,-33.499
C09660=1013.168,29.475,-119.819,-27.852,42.534,-33.511
C09661=1013.169,29.240,-119.798,-27.849,42.503,-33.522
C09662=1013.170,29.005,-119.779,-27.846,42.474,-33.532
C09663=1013.171,28.770,-119.758,-27.843,42.444,-33.542
C09664=1013.172,28.534,-119.739,-27.840,42.414,-33.554
C09665=1013.173,28.300,-119.718,-27.837,42.385,-33.564
C09666=1013.175,28.066,-119.698,-27.834,42.355,-33.574
C09667=1013.175,27.832,-119.679,-27.831,42.326,-33.584
C09668=1013.177,27.598,-119.659,-27.828,42.298,-33.594
C09669=1013.178,27.364,-119.639,-27.825,42.270,-33.604
C09670=1013.179,27.130,-119.619,-27.823,42.241,-33.615
C09671=1013.181,26.896,-119.599,-27.820,42.213,-33.624
C09672=1013.181,26.662,-119.579,-27.817,42.185,-33.636
C09673=1013.183,26.426,-119.559,-27.814,42.158,-33.645
C09674=1013.184,26.190,-119.539,-27.811,42.129,-33.656
C09675=1013.185,25.954,-119.519,-27.809,42.102,-33.665
C09676=1013.186,25.716,-119.498,-27.806,42.075,-33.676
C09677=1013.188,25.479,-119.478,-27.803,42.047,-33.685
C09678=1013.188,25.243,-119.458,-27.800,42.021,-33.695
C09679=1013.190,25.007,-119.439,-27.798,41.994,-33.705
C09680=1013.190,24.773,-119.418,-27.795,41.967,-33.715
C09681=1013.192,24.536,-119.397,-27.792,41.941,-33.724
C09682=1013.193,24.300,-119.377,-27.790,41.915,-33.735
C09683=1013.194,24.069,-119.359,-27.787,41.889,-33.744
C09684=1013.195,23.846,-119.339,-27.785,41.865,-33.754
C09685=1013.196,23.637,-119.322,-27.782,41.842,-33.761
C09686=1013.198,23.273,-119.290,-27.779,41.804,-33.777
C09687=1013.199,22.973,-119.265,-27.775,41.771,-33.788
C09688=1013.200,22.681,-119.240,-27.772,41.741,-33.800
C09689=1013.202,22.336,-119.211,-27.768,41.705,-33.813
C09690=1013.203,21.924,-119.176,-27.764,41.662,-33.830
C09691=1013.205,21.513,-119.140,-27.760,41.621,-33.845
C09692=1013.206,21.253,-119.119,-27.757,41.596,-33.856
C09693=1013.208,20.964,-119.094,-27.754,41.567,-33.867
C09694=1013.209,20.655,-119.068,-27.751,41.537,-33.879
C09695=1013.210,20.335,-119.040,-27.748,41.505,-33.891
C09696=1013.212,20.017,-119.014,-27.745,41.475,-33.903
C09697=1013.213,19.718,-118.988,-27.742,41.447,-33.914
C09698=1013.214,19.321,-118.954,-27.738,41.410,-33.929
C09699=1013.216,19.017,-118.929,-27.735,41.382,-33.941
C09700=1013.217,18.755,-118.906,-27.733,41.357,-33.950
C09701=1013.217,18.522,-118.886,-27.730,41.336,-33.959
C09702=1013.218,18.288,-118.867,-27.728,41.315,-33.967
C09703=1013.219,18.056,-118.847,-27.726,41.296,-33.975
C09704=1013.221,17.823,-118.827,-27.724,41.275,-33.983
C09705=1013.222,17.591,-118.807,-27.722,41.254,-33.992
C09706=1013.222,17.360,-118.788,-27.720,41.235,-34.000
C09707=1013.223,17.129,-118.768,-27.718,41.216,-34.008
C09708=1013.224,16.900,-118.748,-27.716,41.197,-34.015
C09709=1013.225,16.671,-118.729,-27.714,41.178,-34.023
C09710=1013.225,16.442,-118.710,-27.712,41.158,-34.031
C09711=1013.226,16.215,-118.691,-27.710,41.140,-34.039
C09712=1013.227,15.988,-118.671,-27.708,41.121,-34.047
C09713=1013.228,15.761,-118.652,-27.706,41.103,-34.054
C09714=1013.229,15.533,-118.632,-27.704,41.085,-34.063
C09715=1013.230,15.307,-118.614,-27.702,41.067,-34.070
C09716=1013.230,15.081,-118.595,-27.701,41.051,-34.077
C09717=1013.231,14.856,-118.575,-27.699,41.033,-34.084
C09718=1013.232,14.629,-118.556,-27.697,41.015,-34.093
C09719=1013.233,14.403,-118.536,-27.695,40.999,-34.099
C09720=1013.234,14.177,-118.518,-27.693,40.982,-34.107
C09721=1013.234,13.950,-118.498,-27.692,40.965,-34.114
C09722=1013.235,13.723,-118.479,-27.690,40.949,-34.122
C09723=1013.235,13.496,-118.459,-27.688,40.933,-34.128
C09724=1013.236,13.269,-118.440,-27.687,40.916,-34.136
C09725=1013.237,13.040,-118.421,-27.685,40.900,-34.142
C09726=1013.238,12.812,-118.402,-27.683,40.885,-34.151
C09727=1013.239,12.584,-118.383,-27.682,40.869,-34.157
C09728=1013.239,12.355,-118.363,-27.680,40.854,-34.164
C09729=1013.240,12.126,-118.344,-27.678,40.839,-34.171
C09730=1013.241,11.900,-118.325,-27.677,40.824,-34.178
C09731=1013.242,11.676,-118.306,-27.675,40.809,-34.184
C09732=1013.242,11.457,-118.287,-27.674,40.794,-34.190
C09733=1013.243,11.241,-118.269,-27.672,40.781,-34.196
C09734=1013.243,11.025,-118.251,-27.671,40.767,-34.204
C09735=1013.244,10.808,-118.233,-27.669,40.754,-34.210
C09736=1013.245,10.587,-118.213,-27.668,40.740,-34.216
C09737=1013.245,10.362,-118.195,-27.667,40.727,-34.222
C09738=1013.246,10.138,-118.175,-27.665,40.713,-34.228
C09739=1013.247,9.913,-118.157,-27.664,40.700,-34.234
C09740=1013.247,9.689,-118.138,-27.662,40.688,-34.241
C09741=1013.248,9.467,-118.119,-27.661,40.674,-34.247
C09742=1013.249,9.244,-118.100,-27.660,40.663,-34.253
C09743=1013.249,9.021,-118.081,-27.659,40.650,-34.259
C09744=1013.250,8.799,-118.062,-27.657,40.639,-34.265
C09745=1013.250,8.577,-118.043,-27.656,40.626,-34.271
C09746=1013.251,8.354,-118.024,-27.655,40.614,-34.277
C09747=1013.252,8.131,-118.005,-27.654,40.603,-34.282
C09748=1013.252,7.908,-117.986,-27.652,40.592,-34.288
C09749=1013.252,7.683,-117.968,-27.651,40.580,-34.294
C09750=1013.253,7.458,-117.948,-27.650,40.569,-34.300
C09751=1013.254,7.232,-117.930,-27.649,40.559,-34.306
C09752=1013.254,7.005,-117.910,-27.648,40.548,-34.312
C09753=1013.254,6.776,-117.891,-27.647,40.536,-34.317
C09754=1013.255,6.545,-117.872,-27.645,40.526,-34.322
C09755=1013.256,6.312,-117.851,-27.644,40.516,-34.328
C09756=1013.256,6.078,-117.832,-27.643,40.505,-34.334
C09757=1013.257,5.844,-117.812,-27.642,40.495,-34.339
C09758=1013.258,5.610,-117.793,-27.641,40.485,-34.345
C09759=1013.258,5.377,-117.772,-27.640,40.475,-34.350
C09760=1013.258,5.145,-117.753,-27.639,40.466,-34.355
C09761=1013.259,4.913,-117.733,-27.638,40.457,-34.360
C09762=1013.260,4.682,-117.714,-27.637,40.448,-34.366
C09763=1013.260,4.451,-117.695,-27.636,40.439,-34.371
C09764=1013.261,4.218,-117.675,-27.636,40.431,-34.377
C09765=1013.261,3.985,-117.655,-27.635,40.422,-34.380
C09766=1013.261,3.757,-117.636,-27.634,40.414,-34.386
C09767=1013.262,3.538,-117.618,-27.633,40.406,-34.391
C09768=1013.263,3.330,-117.600,-27.632,40.400,-34.394
C09769=1013.263,2.938,-117.566,-27.631,40.386,-34.402
C09770=1013.264,2.555,-117.534,-27.630,40.375,-34.411
C09771=1013.265,2.145,-117.500,-27.629,40.362,-34.418
C09772=1013.265,1.925,-117.482,-27.628,40.356,-34.423
C09773=1013.265,1.696,-117.462,-27.627,40.350,-34.427
C09774=1013.266,1.462,-117.443,-27.627,40.343,-34.432
C09775=1013.266,1.225,-117.422,-27.626,40.338,-34.435
C09776=1013.266,0.989,-117.402,-27.626,40.332,-34.441
C09777=1013.266,0.753,-117.383,-27.625,40.326,-34.445
C09778=1013.267,0.518,-117.363,-27.625,40.321,-34.449
C09779=1013.268,0.283,-117.343,-27.624,40.315,-34.453
C09780=1013.268,0.049,-117.323,-27.624,40.310,-34.457
C09781=1013.268,-0.187,-117.304,-27.623,40.305,-34.461
C09782=1013.269,-0.423,-117.284,-27.623,40.301,-34.464
C09783=1013.269,-0.662,-117.264,-27.622,40.296,-34.468
C09784=1013.270,-0.899,-117.243,-27.622,40.293,-34.472
C09785=1013.269,-1.139,-117.223,-27.621,40.288,-34.476
C09786=1013.269,-1.379,-117.203,-27.621,40.285,-34.480
C09787=1013.271,-1.619,-117.183,-27.621,40.282,-34.483
C09788=1013.271,-1.861,-117.163,-27.621,40.278,-34.486
C09789=1013.271,-2.103,-117.142,-27.620,40.275,-34.490
C09790=1013.271,-2.346,-117.122,-27.620,40.273,-34.494
C09791=1013.272,-2.588,-117.101,-27.620,40.269,-34.498
C09792=1013.272,-2.832,-117.082,-27.620,40.267,-34.502
C09793=1013.272,-3.077,-117.060,-27.620,40.264,-34.504
C09794=1013.273,-3.321,-117.039,-27.619,40.263,-34.506
C09795=1013.273,-3.564,-117.019,-27.619,40.260,-34.511
C09796=1013.272,-3.801,-116.999,-27.619,40.260,-34.514
C09797=1013.273,-4.032,-116.980,-27.619,40.258,-34.517
C09798=1013.273,-4.258,-116.961,-27.619,40.256,-34.519
C09799=1013.273,-4.483,-116.943,-27.619,40.256,-34.521
C09800=1013.273,-4.712,-116.923,-27.619,40.256,-34.525
C09801=1013.274,-4.947,-116.904,-27.619,40.255,-34.528
C09802=1013.274,-5.191,-116.882,-27.619,40.255,-34.530
C09803=1013.274,-5.444,-116.862,-27.620,40.256,-34.532
C09804=1013.274,-5.700,-116.840,-27.620,40.255,-34.536
C09805=1013.275,-5.958,-116.818,-27.620,40.256,-34.538
C09806=1013.275,-6.216,-116.796,-27.620,40.257,-34.541
C09807=1013.275,-6.475,-116.775,-27.620,40.258,-34.543
C09808=1013.275,-6.732,-116.753,-27.621,40.260,-34.544
C09809=1013.276,-6.989,-116.732,-27.621,40.261,-34.548
C09810=1013.275,-7.245,-116.710,-27.621,40.263,-34.549
C09811=1013.275,-7.500,-116.689,-27.622,40.265,-34.552
C09812=1013.275,-7.754,-116.667,-27.622,40.267,-34.554
C09813=1013.276,-8.007,-116.646,-27.622,40.270,-34.555
C09814=1013.276,-8.260,-116.625,-27.623,40.273,-34.558
C09815=1013.275,-8.512,-116.604,-27.623,40.276,-34.560
C09816=1013.275,-8.763,-116.583,-27.624,40.280,-34.561
C09817=1013.276,-9.014,-116.562,-27.624,40.283,-34.562
C09818=1013.276,-9.266,-116.541,-27.625,40.287,-34.563
C09819=1013.276,-9.517,-116.520,-27.626,40.291,-34.566
C09820=1013.276,-9.768,-116.499,-27.626,40.296,-34.567
C09821=1013.275,-10.018,-116.477,-27.627,40.300,-34.568
C09822=1013.276,-10.270,-116.457,-27.628,40.305,-34.570
C09823=1013.277,-10.519,-116.436,-27.628,40.310,-34.571
C09824=1013.276,-10.769,-116.414,-27.629,40.316,-34.572
C09825=1013.276,-11.019,-116.394,-27.630,40.321,-34.573
C09826=1013.276,-11.267,-116.373,-27.631,40.327,-34.574
C09827=1013.276,-11.516,-116.352,-27.632,40.334,-34.574
C09828=1013.276,-11.763,-116.332,-27.632,40.340,-34.575
C09829=1013.276,-12.011,-116.310,-27.633,40.346,-34.575
C09830=1013.276,-12.258,-116.290,-27.634,40.353,-34.576
C09831=1013.276,-12.504,-116.269,-27.635,40.360,-34.577
C09832=1013.276,-12.751,-116.249,-27.636,40.367,-34.578
C09833=1013.276,-12.994,-116.228,-27.637,40.375,-34.578
C09834=1013.276,-13.235,-116.208,-27.638,40.383,-34.577
C09835=1013.276,-13.473,-116.188,-27.639,40.390,-34.577
C09836=1013.275,-13.706,-116.169,-27.640,40.398,-34.578
C09837=1013.276,-13.935,-116.149,-27.641,40.405,-34.578
C09838=1013.275,-14.161,-116.130,-27.642,40.414,-34.578
C09839=1013.275,-14.385,-116.112,-27.643,40.422,-34.578
C09840=1013.275,-14.607,-116.094,-27.644,40.430,-34.579
C09841=1013.275,-14.831,-116.074,-27.646,40.438,-34.579
C09842=1013.274,-15.055,-116.056,-27.647,40.448,-34.578
C09843=1013.275,-15.282,-116.038,-27.648,40.457,-34.579
C09844=1013.274,-15.512,-116.018,-27.649,40.465,-34.579
C09845=1013.274,-15.745,-115.998,-27.650,40.475,-34.578
C09846=1013.275,-15.980,-115.979,-27.652,40.486,-34.577
C09847=1013.274,-16.216,-115.959,-27.653,40.497,-34.576
C09848=1013.274,-16.451,-115.939,-27.654,40.507,-34.575
C09849=1013.274,-16.686,-115.920,-27.656,40.518,-34.575
C09850=1013.274,-16.923,-115.900,-27.657,40.529,-34.573
C09851=1013.273,-17.161,-115.880,-27.659,40.540,-34.573
C09852=1013.273,-17.395,-115.861,-27.660,40.552,-34.571
C09853=1013.273,-17.625,-115.841,-27.662,40.564,-34.570
C09854=1013.273,-17.857,-115.822,-27.663,40.576,-34.570
C09855=1013.272,-18.104,-115.801,-27.665,40.589,-34.568
C09856=1013.273,-18.389,-115.778,-27.667,40.603,-34.567
C09857=1013.271,-18.706,-115.751,-27.669,40.621,-34.565
C09858=1013.271,-19.038,-115.724,-27.671,40.639,-34.563
C09859=1013.271,-19.363,-115.697,-27.674,40.657,-34.562
C09860=1013.271,-19.662,-115.671,-27.676,40.676,-34.559
C09861=1013.270,-19.923,-115.649,-27.678,40.691,-34.558
C09862=1013.270,-20.273,-115.621,-27.680,40.712,-34.554
C09863=1013.269,-20.550,-115.598,-27.683,40.729,-34.552
C09864=1013.270,-20.784,-115.578,-27.685,40.744,-34.551
C09865=1013.269,-21.018,-115.559,-27.686,40.760,-34.548
C09866=1013.269,-21.253,-115.539,-27.688,40.775,-34.547
C09867=1013.268,-21.486,-115.519,-27.690,40.791,-34.545
C09868=1013.268,-21.721,-115.500,-27.692,40.807,-34.542
C09869=1013.267,-21.955,-115.480,-27.694,40.823,-34.540
C09870=1013.267,-22.189,-115.461,-27.696,40.838,-34.538
C09871=1013.266,-22.423,-115.442,-27.698,40.854,-34.535
C09872=1013.266,-22.657,-115.421,-27.700,40.871,-34.533
C09873=1013.266,-22.891,-115.402,-27.703,40.889,-34.530
C09874=1013.265,-23.125,-115.383,-27.705,40.906,-34.529
C09875=1013.265,-23.359,-115.364,-27.707,40.923,-34.525
C09876=1013.264,-23.593,-115.344,-27.709,40.941,-34.522
C09877=1013.264,-23.827,-115.324,-27.711,40.958,-34.519
C09878=1013.264,-24.061,-115.305,-27.713,40.977,-34.517
C09879=1013.263,-24.295,-115.285,-27.716,40.995,-34.514
C09880=1013.263,-24.530,-115.266,-27.718,41.015,-34.510
C09881=1013.262,-24.764,-115.247,-27.720,41.033,-34.508
C09882=1013.262,-24.997,-115.227,-27.723,41.052,-34.504
C09883=1013.261,-25.231,-115.208,-27.725,41.071,-34.501
C09884=1013.261,-25.465,-115.188,-27.728,41.091,-34.498
C09885=1013.261,-25.700,-115.169,-27.730,41.111,-34.495
C09886=1013.260,-25.934,-115.149,-27.733,41.131,-34.492
C09887=1013.259,-26.168,-115.129,-27.735,41.151,-34.488
C09888=1013.259,-26.402,-115.110,-27.738,41.172,-34.484
C09889=1013.258,-26.636,-115.091,-27.740,41.192,-34.480
C09890=1013.258,-26.870,-115.072,-27.743,41.214,-34.476
C09891=1013.257,-27.104,-115.052,-27.745,41.235,-34.474
C09892=1013.257,-27.338,-115.032,-27.748,41.256,-34.469
C09893=1013.256,-27.572,-115.013,-27.750,41.278,-34.465
C09894=1013.256,-27.807,-114.993,-27.753,41.301,-34.462
C09895=1013.255,-28.041,-114.974,-27.756,41.323,-34.457
C09896=1013.255,-28.275,-114.955,-27.759,41.346,-34.453
C09897=1013.254,-28.509,-114.935,-27.761,41.368,-34.449
C09898=1013.253,-28.743,-114.915,-27.764,41.391,-34.444
C09899=1013.253,-28.977,-114.896,-27.767,41.415,-34.440
C09900=1013.252,-29.211,-114.877,-27.770,41.439,-34.436
C09901=1013.251,-29.446,-114.857,-27.773,41.462,-34.431
C09902=1013.251,-29.680,-114.838,-27.776,41.487,-34.427
C09903=1013.250,-29.914,-114.818,-27.779,41.510,-34.422
C09904=1013.250,-30.148,-114.799,-27.782,41.535,-34.418
C09905=1013.249,-30.382,-114.780,-27.785,41.560,-34.413
C09906=1013.248,-30.617,-114.760,-27.788,41.585,-34.409
C09907=1013.247,-30.851,-114.741,-27.791,41.610,-34.404
C09908=1013.247,-31.085,-114.722,-27.794,41.636,-34.399
C09909=1013.246,-31.319,-114.702,-27.797,41.661,-34.393
C09910=1013.246,-31.553,-114.682,-27.800,41.687,-34.389
C09911=1013.245,-31.788,-114.663,-27.803,41.713,-34.384
C09912=1013.244,-32.022,-114.644,-27.806,41.741,-34.378
C09913=1013.244,-32.256,-114.624,-27.810,41.767,-34.373
C09914=1013.243,-32.490,-114.605,-27.813,41.794,-34.368
C09915=1013.242,-32.724,-114.585,-27.816,41.822,-34.362
C09916=1013.241,-32.958,-114.565,-27.819,41.849,-34.356
C09917=1013.241,-33.192,-114.546,-27.823,41.877,-34.351
C09918=1013.240,-33.427,-114.527,-27.826,41.905,-34.346
C09919=1013.239,-33.661,-114.507,-27.829,41.933,-34.340
C09920=1013.239,-33.896,-114.488,-27.833,41.962,-34.334
C09921=1013.238,-34.129,-114.468,-27.836,41.990,-34.329
C09922=1013.237,-34.363,-114.450,-27.840,42.020,-34.323
C09923=1013.235,-34.598,-114.430,-27.843,42.049,-34.316
C09924=1013.235,-34.832,-114.411,-27.847,42.078,-34.310
C09925=1013.234,-35.066,-114.392,-27.850,42.108,-34.305
C09926=1013.234,-35.299,-114.372,-27.854,42.139,-34.299
C09927=1013.233,-35.534,-114.352,-27.857,42.169,-34.293
C09928=1013.232,-35.768,-114.333,-27.861,42.200,-34.286
C09929=1013.232,-36.003,-114.313,-27.865,42.230,-34.281
C09930=1013.230,-36.237,-114.294,-27.868,42.261,-34.274
C09931=1013.229,-36.471,-114.275,-27.872,42.293,-34.268
C09932=1013.228,-36.705,-114.255,-27.876,42.325,-34.261
C09933=1013.228,-36.939,-114.236,-27.880,42.356,-34.255
C09934=1013.227,-37.174,-114.216,-27.883,42.389,-34.247
C09935=1013.226,-37.408,-114.197,-27.887,42.421,-34.241
C09936=1013.225,-37.641,-114.178,-27.891,42.453,-34.235
C09937=1013.224,-37.876,-114.158,-27.895,42.486,-34.228
C09938=1013.223,-38.110,-114.139,-27.899,42.520,-34.221
C09939=1013.223,-38.344,-114.120,-27.903,42.553,-34.214
C09940=1013.221,-38.578,-114.099,-27.906,42.587,-34.207
C09941=1013.220,-38.812,-114.081,-27.910,42.620,-34.200
C09942=1013.219,-39.046,-114.062,-27.914,42.655,-34.193
C09943=1013.219,-39.281,-114.042,-27.918,42.690,-34.186
C09944=1013.218,-39.515,-114.022,-27.923,42.725,-34.178
C09945=1013.216,-39.749,-114.003,-27.927,42.759,-34.172
C09946=1013.216,-39.983,-113.984,-27.931,42.794,-34.164
C09947=1013.215,-40.218,-113.965,-27.935,42.830,-34.156
C09948=1013.213,-40.451,-113.945,-27.939,42.866,-34.149
C09949=1013.213,-40.685,-113.926,-27.943,42.902,-34.141
C09950=1013.212,-40.919,-113.907,-27.947,42.938,-34.134
C09951=1013.210,-41.153,-113.887,-27.951,42.974,-34.127
C09952=1013.210,-41.387,-113.868,-27.956,43.011,-34.118
C09953=1013.209,-41.621,-113.848,-27.960,43.049,-34.111
C09954=1013.207,-41.855,-113.829,-27.964,43.087,-34.103
C09955=1013.206,-42.089,-113.810,-27.969,43.124,-34.095
C09956=1013.206,-42.323,-113.790,-27.973,43.161,-34.087
C09957=1013.204,-42.557,-113.771,-27.977,43.200,-34.080
C09958=1013.203,-42.791,-113.751,-27.982,43.238,-34.071
C09959=1013.203,-43.026,-113.732,-27.986,43.278,-34.062
C09960=1013.201,-43.259,-113.713,-27.991,43.316,-34.055
C09961=1013.201,-43.493,-113.694,-27.995,43.355,-34.047
C09962=1013.199,-43.727,-113.674,-28.000,43.395,-34.039
C09963=1013.198,-43.961,-113.655,-28.004,43.434,-34.030
C09964=1013.197,-44.195,-113.636,-28.009,43.475,-34.021
C09965=1013.196,-44.428,-113.616,-28.013,43.515,-34.013
C09966=1013.194,-44.663,-113.597,-28.018,43.556,-34.004
C09967=1013.193,-44.896,-113.577,-28.023,43.596,-33.996
C09968=1013.192,-45.130,-113.558,-28.027,43.638,-33.988
C09969=1013.192,-45.364,-113.539,-28.032,43.679,-33.979
C09970=1013.190,-45.597,-113.520,-28.037,43.720,-33.970
C09971=1013.189,-45.832,-113.500,-28.041,43.762,-33.962
C09972=1013.187,-46.065,-113.481,-28.046,43.805,-33.952
C09973=1013.187,-46.300,-113.462,-28.051,43.847,-33.944
C09974=1013.185,-46.533,-113.442,-28.056,43.890,-33.934
C09975=1013.185,-46.767,-113.423,-28.061,43.933,-33.925
C09976=1013.183,-47.001,-113.403,-28.065,43.977,-33.916
C09977=1013.182,-47.235,-113.384,-28.070,44.020,-33.907
C09978=1013.181,-47.468,-113.365,-28.075,44.064,-33.898
C09979=1013.179,-47.702,-113.346,-28.080,44.107,-33.889
C09980=1013.179,-47.936,-113.326,-28.085,44.152,-33.880
C09981=1013.177,-48.170,-113.307,-28.090,44.196,-33.871
C09982=1013.176,-48.404,-113.287,-28.095,44.241,-33.861
C09983=1013.175,-48.637,-113.268,-28.100,44.286,-33.851
C09984=1013.173,-48.871,-113.249,-28.105,44.332,-33.842
//INST
///DATE 2021/06/17 16:00
///ATTR SC,RW,RJ
////FRAME USER -1
///GROUP1 RB1
NOP
MOVJ C00000 VJ=100.00 PL=0
'Path Start: Op_ID_1
MOVJ C00001 VJ=25.00 PL=0
MOVJ C00002 VJ=25.00 PL=0
MOVL C00003 V=800.0 PL=0
'CALL JOB: TOOL ON
MOVL C00004 V=800.0 PL=0
MOVL C00005 V=800.0 PL=0
MOVL C00006 V=800.0 PL=0
MOVL C00007 V=800.0 PL=0
MOVL C00008 V=800.0 PL=0
MOVL C00009 V=800.0 PL=0
MOVL C00010 V=800.0 PL=0
MOVL C00011 V=800.0 PL=0
MOVL C00012 V=800.0 PL=0
MOVL C00013 V=800.0 PL=0
MOVL C00014 V=800.0 PL=0
MOVL C00015 V=800.0 PL=0
MOVL C00016 V=800.0 PL=0
MOVL C00017 V=800.0 PL=0
MOVL C00018 V=800.0 PL=0
MOVL C00019 V=800.0 PL=0
MOVL C00020 V=800.0 PL=0
MOVL C00021 V=800.0 PL=0
MOVL C00022 V=800.0 PL=0
MOVL C00023 V=800.0 PL=0
MOVL C00024 V=800.0 PL=0
MOVL C00025 V=800.0 PL=0
MOVL C00026 V=800.0 PL=0
MOVL C00027 V=800.0 PL=0
MOVL C00028 V=800.0 PL=0
MOVL C00029 V=800.0 PL=0
MOVL C00030 V=800.0 PL=0
MOVL C00031 V=800.0 PL=0
MOVL C00032 V=800.0 PL=0
MOVL C00033 V=800.0 PL=0
MOVL C00034 V=800.0 PL=0
MOVL C00035 V=800.0 PL=0
MOVL C00036 V=800.0 PL=0
MOVL C00037 V=800.0 PL=0
MOVL C00038 V=800.0 PL=0
MOVL C00039 V=800.0 PL=0
MOVL C00040 V=800.0 PL=0
MOVL C00041 V=800.0 PL=0
MOVL C00042 V=800.0 PL=0
MOVL C00043 V=800.0 PL=0
MOVL C00044 V=800.0 PL=0
MOVL C00045 V=800.0 PL=0
MOVL C00046 V=800.0 PL=0
MOVL C00047 V=800.0 PL=0
MOVL C00048 V=800.0 PL=0
MOVL C00049 V=800.0 PL=0
MOVL C00050 V=800.0 PL=0
MOVL C00051 V=800.0 PL=0
MOVL C00052 V=800.0 PL=0
MOVL C00053 V=800.0 PL=0
MOVL C00054 V=800.0 PL=0
MOVL C00055 V=800.0 PL=0
MOVL C00056 V=800.0 PL=0
MOVL C00057 V=800.0 PL=0
MOVL C00058 V=800.0 PL=0
MOVL C00059 V=800.0 PL=0
MOVL C00060 V=800.0 PL=0
MOVL C00061 V=800.0 PL=0
MOVL C00062 V=800.0 PL=0
MOVL C00063 V=800.0 PL=0
MOVL C00064 V=800.0 PL=0
MOVL C00065 V=800.0 PL=0
MOVL C00066 V=800.0 PL=0
MOVL C00067 V=800.0 PL=0
MOVL C00068 V=800.0 PL=0
MOVL C00069 V=800.0 PL=0
MOVL C00070 V=800.0 PL=0
MOVL C00071 V=800.0 PL=0
MOVL C00072 V=800.0 PL=0
MOVL C00073 V=800.0 PL=0
MOVL C00074 V=800.0 PL=0
MOVL C00075 V=800.0 PL=0
MOVL C00076 V=800.0 PL=0
MOVL C00077 V=800.0 PL=0
MOVL C00078 V=800.0 PL=0
MOVL C00079 V=800.0 PL=0
MOVL C00080 V=800.0 PL=0
MOVL C00081 V=800.0 PL=0
MOVL C00082 V=800.0 PL=0
MOVL C00083 V=800.0 PL=0
MOVL C00084 V=800.0 PL=0
MOVL C00085 V=800.0 PL=0
MOVL C00086 V=800.0 PL=0
MOVL C00087 V=800.0 PL=0
MOVL C00088 V=800.0 PL=0
MOVL C00089 V=800.0 PL=0
MOVL C00090 V=800.0 PL=0
MOVL C00091 V=800.0 PL=0
MOVL C00092 V=800.0 PL=0
MOVL C00093 V=800.0 PL=0
MOVL C00094 V=800.0 PL=0
MOVL C00095 V=800.0 PL=0
MOVL C00096 V=800.0 PL=0
MOVL C00097 V=800.0 PL=0
MOVL C00098 V=800.0 PL=0
MOVL C00099 V=800.0 PL=0
MOVL C00100 V=800.0 PL=0
MOVL C00101 V=800.0 PL=0
MOVL C00102 V=800.0 PL=0
MOVL C00103 V=800.0 PL=0
MOVL C00104 V=800.0 PL=0
MOVL C00105 V=800.0 PL=0
MOVL C00106 V=800.0 PL=0
MOVL C00107 V=800.0 PL=0
MOVL C00108 V=800.0 PL=0
MOVL C00109 V=800.0 PL=0
MOVL C00110 V=800.0 PL=0
MOVL C00111 V=800.0 PL=0
MOVL C00112 V=800.0 PL=0
MOVL C00113 V=800.0 PL=0
MOVL C00114 V=800.0 PL=0
MOVL C00115 V=800.0 PL=0
MOVL C00116 V=800.0 PL=0
MOVL C00117 V=800.0 PL=0
MOVL C00118 V=800.0 PL=0
MOVL C00119 V=800.0 PL=0
MOVL C00120 V=800.0 PL=0
MOVL C00121 V=800.0 PL=0
MOVL C00122 V=800.0 PL=0
MOVL C00123 V=800.0 PL=0
MOVL C00124 V=800.0 PL=0
MOVL C00125 V=800.0 PL=0
MOVL C00126 V=800.0 PL=0
MOVL C00127 V=800.0 PL=0
MOVL C00128 V=800.0 PL=0
MOVL C00129 V=800.0 PL=0
MOVL C00130 V=800.0 PL=0
MOVL C00131 V=800.0 PL=0
MOVL C00132 V=800.0 PL=0
MOVL C00133 V=800.0 PL=0
MOVL C00134 V=800.0 PL=0
MOVL C00135 V=800.0 PL=0
MOVL C00136 V=800.0 PL=0
MOVL C00137 V=800.0 PL=0
MOVL C00138 V=800.0 PL=0
MOVL C00139 V=800.0 PL=0
MOVL C00140 V=800.0 PL=0
MOVL C00141 V=800.0 PL=0
MOVL C00142 V=800.0 PL=0
MOVL C00143 V=800.0 PL=0
MOVL C00144 V=800.0 PL=0
MOVL C00145 V=800.0 PL=0
MOVL C00146 V=800.0 PL=0
MOVL C00147 V=800.0 PL=0
MOVL C00148 V=800.0 PL=0
MOVL C00149 V=800.0 PL=0
MOVL C00150 V=800.0 PL=0
MOVL C00151 V=800.0 PL=0
MOVL C00152 V=800.0 PL=0
MOVL C00153 V=800.0 PL=0
MOVL C00154 V=800.0 PL=0
MOVL C00155 V=800.0 PL=0
MOVL C00156 V=800.0 PL=0
MOVL C00157 V=800.0 PL=0
MOVL C00158 V=800.0 PL=0
MOVL C00159 V=800.0 PL=0
MOVL C00160 V=800.0 PL=0
MOVL C00161 V=800.0 PL=0
MOVL C00162 V=800.0 PL=0
MOVL C00163 V=800.0 PL=0
MOVL C00164 V=800.0 PL=0
MOVL C00165 V=800.0 PL=0
MOVL C00166 V=800.0 PL=0
MOVL C00167 V=800.0 PL=0
MOVL C00168 V=800.0 PL=0
MOVL C00169 V=800.0 PL=0
MOVL C00170 V=800.0 PL=0
MOVL C00171 V=800.0 PL=0
MOVL C00172 V=800.0 PL=0
MOVL C00173 V=800.0 PL=0
MOVL C00174 V=800.0 PL=0
MOVL C00175 V=800.0 PL=0
MOVL C00176 V=800.0 PL=0
MOVL C00177 V=800.0 PL=0
MOVL C00178 V=800.0 PL=0
MOVL C00179 V=800.0 PL=0
MOVL C00180 V=800.0 PL=0
MOVL C00181 V=800.0 PL=0
MOVL C00182 V=800.0 PL=0
MOVL C00183 V=800.0 PL=0
MOVL C00184 V=800.0 PL=0
MOVL C00185 V=800.0 PL=0
MOVL C00186 V=800.0 PL=0
MOVL C00187 V=800.0 PL=0
MOVL C00188 V=800.0 PL=0
MOVL C00189 V=800.0 PL=0
MOVL C00190 V=800.0 PL=0
MOVL C00191 V=800.0 PL=0
MOVL C00192 V=800.0 PL=0
MOVL C00193 V=800.0 PL=0
MOVL C00194 V=800.0 PL=0
MOVL C00195 V=800.0 PL=0
MOVL C00196 V=800.0 PL=0
MOVL C00197 V=800.0 PL=0
MOVL C00198 V=800.0 PL=0
MOVL C00199 V=800.0 PL=0
MOVL C00200 V=800.0 PL=0
MOVL C00201 V=800.0 PL=0
MOVL C00202 V=800.0 PL=0
MOVL C00203 V=800.0 PL=0
MOVL C00204 V=800.0 PL=0
MOVL C00205 V=800.0 PL=0
MOVL C00206 V=800.0 PL=0
MOVL C00207 V=800.0 PL=0
MOVL C00208 V=800.0 PL=0
MOVL C00209 V=800.0 PL=0
MOVL C00210 V=800.0 PL=0
MOVL C00211 V=800.0 PL=0
MOVL C00212 V=800.0 PL=0
MOVL C00213 V=800.0 PL=0
MOVL C00214 V=800.0 PL=0
MOVL C00215 V=800.0 PL=0
MOVL C00216 V=800.0 PL=0
MOVL C00217 V=800.0 PL=0
MOVL C00218 V=800.0 PL=0
MOVL C00219 V=800.0 PL=0
MOVL C00220 V=800.0 PL=0
MOVL C00221 V=800.0 PL=0
MOVL C00222 V=800.0 PL=0
MOVL C00223 V=800.0 PL=0
MOVL C00224 V=800.0 PL=0
MOVL C00225 V=800.0 PL=0
MOVL C00226 V=800.0 PL=0
MOVL C00227 V=800.0 PL=0
MOVL C00228 V=800.0 PL=0
MOVL C00229 V=800.0 PL=0
MOVL C00230 V=800.0 PL=0
MOVL C00231 V=800.0 PL=0
MOVL C00232 V=800.0 PL=0
MOVL C00233 V=800.0 PL=0
MOVL C00234 V=800.0 PL=0
MOVL C00235 V=800.0 PL=0
MOVL C00236 V=800.0 PL=0
MOVL C00237 V=800.0 PL=0
MOVL C00238 V=800.0 PL=0
MOVL C00239 V=800.0 PL=0
MOVL C00240 V=800.0 PL=0
MOVL C00241 V=800.0 PL=0
MOVL C00242 V=800.0 PL=0
MOVL C00243 V=800.0 PL=0
MOVL C00244 V=800.0 PL=0
MOVL C00245 V=800.0 PL=0
MOVL C00246 V=800.0 PL=0
MOVL C00247 V=800.0 PL=0
MOVL C00248 V=800.0 PL=0
MOVL C00249 V=800.0 PL=0
MOVL C00250 V=800.0 PL=0
MOVL C00251 V=800.0 PL=0
MOVL C00252 V=800.0 PL=0
MOVL C00253 V=800.0 PL=0
MOVL C00254 V=800.0 PL=0
MOVL C00255 V=800.0 PL=0
MOVL C00256 V=800.0 PL=0
MOVL C00257 V=800.0 PL=0
MOVL C00258 V=800.0 PL=0
MOVL C00259 V=800.0 PL=0
MOVL C00260 V=800.0 PL=0
MOVL C00261 V=800.0 PL=0
MOVL C00262 V=800.0 PL=0
MOVL C00263 V=800.0 PL=0
MOVL C00264 V=800.0 PL=0
MOVL C00265 V=800.0 PL=0
MOVL C00266 V=800.0 PL=0
MOVL C00267 V=800.0 PL=0
MOVL C00268 V=800.0 PL=0
MOVL C00269 V=800.0 PL=0
MOVL C00270 V=800.0 PL=0
MOVL C00271 V=800.0 PL=0
MOVL C00272 V=800.0 PL=0
MOVL C00273 V=800.0 PL=0
MOVL C00274 V=800.0 PL=0
MOVL C00275 V=800.0 PL=0
MOVL C00276 V=800.0 PL=0
MOVL C00277 V=800.0 PL=0
MOVL C00278 V=800.0 PL=0
MOVL C00279 V=800.0 PL=0
MOVL C00280 V=800.0 PL=0
MOVL C00281 V=800.0 PL=0
MOVL C00282 V=800.0 PL=0
MOVL C00283 V=800.0 PL=0
MOVL C00284 V=800.0 PL=0
MOVL C00285 V=800.0 PL=0
MOVL C00286 V=800.0 PL=0
MOVL C00287 V=800.0 PL=0
MOVL C00288 V=800.0 PL=0
MOVL C00289 V=800.0 PL=0
MOVL C00290 V=800.0 PL=0
MOVL C00291 V=800.0 PL=0
MOVL C00292 V=800.0 PL=0
MOVL C00293 V=800.0 PL=0
MOVL C00294 V=800.0 PL=0
MOVL C00295 V=800.0 PL=0
MOVL C00296 V=800.0 PL=0
MOVL C00297 V=800.0 PL=0
MOVL C00298 V=800.0 PL=0
MOVL C00299 V=800.0 PL=0
MOVL C00300 V=800.0 PL=0
MOVL C00301 V=800.0 PL=0
MOVL C00302 V=800.0 PL=0
MOVL C00303 V=800.0 PL=0
MOVL C00304 V=800.0 PL=0
MOVL C00305 V=800.0 PL=0
MOVL C00306 V=800.0 PL=0
MOVL C00307 V=800.0 PL=0
MOVL C00308 V=800.0 PL=0
MOVL C00309 V=800.0 PL=0
MOVL C00310 V=800.0 PL=0
MOVL C00311 V=800.0 PL=0
MOVL C00312 V=800.0 PL=0
MOVL C00313 V=800.0 PL=0
MOVL C00314 V=800.0 PL=0
MOVL C00315 V=800.0 PL=0
MOVL C00316 V=800.0 PL=0
MOVL C00317 V=800.0 PL=0
MOVL C00318 V=800.0 PL=0
MOVL C00319 V=800.0 PL=0
MOVL C00320 V=800.0 PL=0
MOVL C00321 V=800.0 PL=0
MOVL C00322 V=800.0 PL=0
MOVL C00323 V=800.0 PL=0
MOVL C00324 V=800.0 PL=0
MOVL C00325 V=800.0 PL=0
MOVL C00326 V=800.0 PL=0
MOVL C00327 V=800.0 PL=0
MOVL C00328 V=800.0 PL=0
MOVL C00329 V=800.0 PL=0
MOVL C00330 V=800.0 PL=0
MOVL C00331 V=800.0 PL=0
MOVL C00332 V=800.0 PL=0
MOVL C00333 V=800.0 PL=0
MOVL C00334 V=800.0 PL=0
MOVL C00335 V=800.0 PL=0
MOVL C00336 V=800.0 PL=0
MOVL C00337 V=800.0 PL=0
MOVL C00338 V=800.0 PL=0
MOVL C00339 V=800.0 PL=0
MOVL C00340 V=800.0 PL=0
MOVL C00341 V=800.0 PL=0
MOVL C00342 V=800.0 PL=0
MOVL C00343 V=800.0 PL=0
MOVL C00344 V=800.0 PL=0
MOVL C00345 V=800.0 PL=0
MOVL C00346 V=800.0 PL=0
MOVL C00347 V=800.0 PL=0
MOVL C00348 V=800.0 PL=0
MOVL C00349 V=800.0 PL=0
MOVL C00350 V=800.0 PL=0
MOVL C00351 V=800.0 PL=0
MOVL C00352 V=800.0 PL=0
MOVL C00353 V=800.0 PL=0
MOVL C00354 V=800.0 PL=0
MOVL C00355 V=800.0 PL=0
MOVL C00356 V=800.0 PL=0
MOVL C00357 V=800.0 PL=0
MOVL C00358 V=800.0 PL=0
MOVL C00359 V=800.0 PL=0
MOVL C00360 V=800.0 PL=0
MOVL C00361 V=800.0 PL=0
MOVL C00362 V=800.0 PL=0
MOVL C00363 V=800.0 PL=0
MOVL C00364 V=800.0 PL=0
MOVL C00365 V=800.0 PL=0
MOVL C00366 V=800.0 PL=0
MOVL C00367 V=800.0 PL=0
MOVL C00368 V=800.0 PL=0
MOVL C00369 V=800.0 PL=0
MOVL C00370 V=800.0 PL=0
MOVL C00371 V=800.0 PL=0
MOVL C00372 V=800.0 PL=0
MOVL C00373 V=800.0 PL=0
MOVL C00374 V=800.0 PL=0
MOVL C00375 V=800.0 PL=0
MOVL C00376 V=800.0 PL=0
MOVL C00377 V=800.0 PL=0
MOVL C00378 V=800.0 PL=0
MOVL C00379 V=800.0 PL=0
MOVL C00380 V=800.0 PL=0
MOVL C00381 V=800.0 PL=0
MOVL C00382 V=800.0 PL=0
MOVL C00383 V=800.0 PL=0
MOVL C00384 V=800.0 PL=0
MOVL C00385 V=800.0 PL=0
MOVL C00386 V=800.0 PL=0
MOVL C00387 V=800.0 PL=0
MOVL C00388 V=800.0 PL=0
MOVL C00389 V=800.0 PL=0
MOVL C00390 V=800.0 PL=0
MOVL C00391 V=800.0 PL=0
MOVL C00392 V=800.0 PL=0
MOVL C00393 V=800.0 PL=0
MOVL C00394 V=800.0 PL=0
MOVL C00395 V=800.0 PL=0
MOVL C00396 V=800.0 PL=0
MOVL C00397 V=800.0 PL=0
MOVL C00398 V=800.0 PL=0
MOVL C00399 V=800.0 PL=0
MOVL C00400 V=800.0 PL=0
MOVL C00401 V=800.0 PL=0
MOVL C00402 V=800.0 PL=0
MOVL C00403 V=800.0 PL=0
MOVL C00404 V=800.0 PL=0
MOVL C00405 V=800.0 PL=0
MOVL C00406 V=800.0 PL=0
MOVL C00407 V=800.0 PL=0
MOVL C00408 V=800.0 PL=0
MOVL C00409 V=800.0 PL=0
MOVL C00410 V=800.0 PL=0
MOVL C00411 V=800.0 PL=0
MOVL C00412 V=800.0 PL=0
MOVL C00413 V=800.0 PL=0
MOVL C00414 V=800.0 PL=0
MOVL C00415 V=800.0 PL=0
MOVL C00416 V=800.0 PL=0
MOVL C00417 V=800.0 PL=0
MOVL C00418 V=800.0 PL=0
MOVL C00419 V=800.0 PL=0
MOVL C00420 V=800.0 PL=0
MOVL C00421 V=800.0 PL=0
MOVL C00422 V=800.0 PL=0
MOVL C00423 V=800.0 PL=0
MOVL C00424 V=800.0 PL=0
MOVL C00425 V=800.0 PL=0
MOVL C00426 V=800.0 PL=0
MOVL C00427 V=800.0 PL=0
MOVL C00428 V=800.0 PL=0
MOVL C00429 V=800.0 PL=0
MOVL C00430 V=800.0 PL=0
MOVL C00431 V=800.0 PL=0
MOVL C00432 V=800.0 PL=0
MOVL C00433 V=800.0 PL=0
MOVL C00434 V=800.0 PL=0
MOVL C00435 V=800.0 PL=0
MOVL C00436 V=800.0 PL=0
MOVL C00437 V=800.0 PL=0
MOVL C00438 V=800.0 PL=0
MOVL C00439 V=800.0 PL=0
MOVL C00440 V=800.0 PL=0
MOVL C00441 V=800.0 PL=0
MOVL C00442 V=800.0 PL=0
MOVL C00443 V=800.0 PL=0
MOVL C00444 V=800.0 PL=0
MOVL C00445 V=800.0 PL=0
MOVL C00446 V=800.0 PL=0
MOVL C00447 V=800.0 PL=0
MOVL C00448 V=800.0 PL=0
MOVL C00449 V=800.0 PL=0
MOVL C00450 V=800.0 PL=0
MOVL C00451 V=800.0 PL=0
MOVL C00452 V=800.0 PL=0
MOVL C00453 V=800.0 PL=0
MOVL C00454 V=800.0 PL=0
MOVL C00455 V=800.0 PL=0
MOVL C00456 V=800.0 PL=0
MOVL C00457 V=800.0 PL=0
MOVL C00458 V=800.0 PL=0
MOVL C00459 V=800.0 PL=0
MOVL C00460 V=800.0 PL=0
MOVL C00461 V=800.0 PL=0
MOVL C00462 V=800.0 PL=0
MOVL C00463 V=800.0 PL=0
MOVL C00464 V=800.0 PL=0
MOVL C00465 V=800.0 PL=0
MOVL C00466 V=800.0 PL=0
MOVL C00467 V=800.0 PL=0
MOVL C00468 V=800.0 PL=0
MOVL C00469 V=800.0 PL=0
MOVL C00470 V=800.0 PL=0
MOVL C00471 V=800.0 PL=0
MOVL C00472 V=800.0 PL=0
MOVL C00473 V=800.0 PL=0
MOVL C00474 V=800.0 PL=0
MOVL C00475 V=800.0 PL=0
MOVL C00476 V=800.0 PL=0
MOVL C00477 V=800.0 PL=0
MOVL C00478 V=800.0 PL=0
MOVL C00479 V=800.0 PL=0
MOVL C00480 V=800.0 PL=0
MOVL C00481 V=800.0 PL=0
MOVL C00482 V=800.0 PL=0
MOVL C00483 V=800.0 PL=0
MOVL C00484 V=800.0 PL=0
MOVL C00485 V=800.0 PL=0
MOVL C00486 V=800.0 PL=0
MOVL C00487 V=800.0 PL=0
MOVL C00488 V=800.0 PL=0
MOVL C00489 V=800.0 PL=0
MOVL C00490 V=800.0 PL=0
MOVL C00491 V=800.0 PL=0
MOVL C00492 V=800.0 PL=0
MOVL C00493 V=800.0 PL=0
MOVL C00494 V=800.0 PL=0
MOVL C00495 V=800.0 PL=0
MOVL C00496 V=800.0 PL=0
MOVL C00497 V=800.0 PL=0
MOVL C00498 V=800.0 PL=0
MOVL C00499 V=800.0 PL=0
MOVL C00500 V=800.0 PL=0
MOVL C00501 V=800.0 PL=0
MOVL C00502 V=800.0 PL=0
MOVL C00503 V=800.0 PL=0
MOVL C00504 V=800.0 PL=0
MOVL C00505 V=800.0 PL=0
MOVL C00506 V=800.0 PL=0
MOVL C00507 V=800.0 PL=0
MOVL C00508 V=800.0 PL=0
MOVL C00509 V=800.0 PL=0
MOVL C00510 V=800.0 PL=0
MOVL C00511 V=800.0 PL=0
MOVL C00512 V=800.0 PL=0
MOVL C00513 V=800.0 PL=0
MOVL C00514 V=800.0 PL=0
MOVL C00515 V=800.0 PL=0
MOVL C00516 V=800.0 PL=0
MOVL C00517 V=800.0 PL=0
MOVL C00518 V=800.0 PL=0
MOVL C00519 V=800.0 PL=0
MOVL C00520 V=800.0 PL=0
MOVL C00521 V=800.0 PL=0
MOVL C00522 V=800.0 PL=0
MOVL C00523 V=800.0 PL=0
MOVL C00524 V=800.0 PL=0
MOVL C00525 V=800.0 PL=0
MOVL C00526 V=800.0 PL=0
MOVL C00527 V=800.0 PL=0
MOVL C00528 V=800.0 PL=0
MOVL C00529 V=800.0 PL=0
MOVL C00530 V=800.0 PL=0
MOVL C00531 V=800.0 PL=0
MOVL C00532 V=800.0 PL=0
MOVL C00533 V=800.0 PL=0
MOVL C00534 V=800.0 PL=0
MOVL C00535 V=800.0 PL=0
MOVL C00536 V=800.0 PL=0
MOVL C00537 V=800.0 PL=0
MOVL C00538 V=800.0 PL=0
MOVL C00539 V=800.0 PL=0
MOVL C00540 V=800.0 PL=0
MOVL C00541 V=800.0 PL=0
MOVL C00542 V=800.0 PL=0
MOVL C00543 V=800.0 PL=0
MOVL C00544 V=800.0 PL=0
MOVL C00545 V=800.0 PL=0
MOVL C00546 V=800.0 PL=0
MOVL C00547 V=800.0 PL=0
MOVL C00548 V=800.0 PL=0
MOVL C00549 V=800.0 PL=0
MOVL C00550 V=800.0 PL=0
MOVL C00551 V=800.0 PL=0
MOVL C00552 V=800.0 PL=0
MOVL C00553 V=800.0 PL=0
MOVL C00554 V=800.0 PL=0
MOVL C00555 V=800.0 PL=0
MOVL C00556 V=800.0 PL=0
MOVL C00557 V=800.0 PL=0
MOVL C00558 V=800.0 PL=0
MOVL C00559 V=800.0 PL=0
MOVL C00560 V=800.0 PL=0
MOVL C00561 V=800.0 PL=0
MOVL C00562 V=800.0 PL=0
MOVL C00563 V=800.0 PL=0
MOVL C00564 V=800.0 PL=0
MOVL C00565 V=800.0 PL=0
MOVL C00566 V=800.0 PL=0
MOVL C00567 V=800.0 PL=0
MOVL C00568 V=800.0 PL=0
MOVL C00569 V=800.0 PL=0
MOVL C00570 V=800.0 PL=0
MOVL C00571 V=800.0 PL=0
MOVL C00572 V=800.0 PL=0
MOVL C00573 V=800.0 PL=0
MOVL C00574 V=800.0 PL=0
MOVL C00575 V=800.0 PL=0
MOVL C00576 V=800.0 PL=0
MOVL C00577 V=800.0 PL=0
MOVL C00578 V=800.0 PL=0
MOVL C00579 V=800.0 PL=0
MOVL C00580 V=800.0 PL=0
MOVL C00581 V=800.0 PL=0
MOVL C00582 V=800.0 PL=0
MOVL C00583 V=800.0 PL=0
MOVL C00584 V=800.0 PL=0
MOVL C00585 V=800.0 PL=0
MOVL C00586 V=800.0 PL=0
MOVL C00587 V=800.0 PL=0
MOVL C00588 V=800.0 PL=0
MOVL C00589 V=800.0 PL=0
MOVL C00590 V=800.0 PL=0
MOVL C00591 V=800.0 PL=0
MOVL C00592 V=800.0 PL=0
MOVL C00593 V=800.0 PL=0
MOVL C00594 V=800.0 PL=0
MOVL C00595 V=800.0 PL=0
MOVL C00596 V=800.0 PL=0
MOVL C00597 V=800.0 PL=0
MOVL C00598 V=800.0 PL=0
MOVL C00599 V=800.0 PL=0
MOVL C00600 V=800.0 PL=0
MOVL C00601 V=800.0 PL=0
MOVL C00602 V=800.0 PL=0
MOVL C00603 V=800.0 PL=0
MOVL C00604 V=800.0 PL=0
MOVL C00605 V=800.0 PL=0
MOVL C00606 V=800.0 PL=0
MOVL C00607 V=800.0 PL=0
MOVL C00608 V=800.0 PL=0
MOVL C00609 V=800.0 PL=0
MOVL C00610 V=800.0 PL=0
MOVL C00611 V=800.0 PL=0
MOVL C00612 V=800.0 PL=0
MOVL C00613 V=800.0 PL=0
MOVL C00614 V=800.0 PL=0
MOVL C00615 V=800.0 PL=0
MOVL C00616 V=800.0 PL=0
MOVL C00617 V=800.0 PL=0
MOVL C00618 V=800.0 PL=0
MOVL C00619 V=800.0 PL=0
MOVL C00620 V=800.0 PL=0
MOVL C00621 V=800.0 PL=0
MOVL C00622 V=800.0 PL=0
MOVL C00623 V=800.0 PL=0
MOVL C00624 V=800.0 PL=0
MOVL C00625 V=800.0 PL=0
MOVL C00626 V=800.0 PL=0
MOVL C00627 V=800.0 PL=0
MOVL C00628 V=800.0 PL=0
MOVL C00629 V=800.0 PL=0
MOVL C00630 V=800.0 PL=0
MOVL C00631 V=800.0 PL=0
MOVL C00632 V=800.0 PL=0
MOVL C00633 V=800.0 PL=0
MOVL C00634 V=800.0 PL=0
MOVL C00635 V=800.0 PL=0
MOVL C00636 V=800.0 PL=0
MOVL C00637 V=800.0 PL=0
MOVL C00638 V=800.0 PL=0
MOVL C00639 V=800.0 PL=0
MOVL C00640 V=800.0 PL=0
MOVL C00641 V=800.0 PL=0
MOVL C00642 V=800.0 PL=0
MOVL C00643 V=800.0 PL=0
MOVL C00644 V=800.0 PL=0
MOVL C00645 V=800.0 PL=0
MOVL C00646 V=800.0 PL=0
MOVL C00647 V=800.0 PL=0
MOVL C00648 V=800.0 PL=0
MOVL C00649 V=800.0 PL=0
MOVL C00650 V=800.0 PL=0
MOVL C00651 V=800.0 PL=0
MOVL C00652 V=800.0 PL=0
MOVL C00653 V=800.0 PL=0
MOVL C00654 V=800.0 PL=0
MOVL C00655 V=800.0 PL=0
MOVL C00656 V=800.0 PL=0
MOVL C00657 V=800.0 PL=0
MOVL C00658 V=800.0 PL=0
MOVL C00659 V=800.0 PL=0
MOVL C00660 V=800.0 PL=0
MOVL C00661 V=800.0 PL=0
MOVL C00662 V=800.0 PL=0
MOVL C00663 V=800.0 PL=0
MOVL C00664 V=800.0 PL=0
MOVL C00665 V=800.0 PL=0
MOVL C00666 V=800.0 PL=0
MOVL C00667 V=800.0 PL=0
MOVL C00668 V=800.0 PL=0
MOVL C00669 V=800.0 PL=0
MOVL C00670 V=800.0 PL=0
MOVL C00671 V=800.0 PL=0
MOVL C00672 V=800.0 PL=0
MOVL C00673 V=800.0 PL=0
MOVL C00674 V=800.0 PL=0
MOVL C00675 V=800.0 PL=0
MOVL C00676 V=800.0 PL=0
MOVL C00677 V=800.0 PL=0
MOVL C00678 V=800.0 PL=0
MOVL C00679 V=800.0 PL=0
MOVL C00680 V=800.0 PL=0
MOVL C00681 V=800.0 PL=0
MOVL C00682 V=800.0 PL=0
MOVL C00683 V=800.0 PL=0
MOVL C00684 V=800.0 PL=0
MOVL C00685 V=800.0 PL=0
MOVL C00686 V=800.0 PL=0
MOVL C00687 V=800.0 PL=0
MOVL C00688 V=800.0 PL=0
MOVL C00689 V=800.0 PL=0
MOVL C00690 V=800.0 PL=0
MOVL C00691 V=800.0 PL=0
MOVL C00692 V=800.0 PL=0
MOVL C00693 V=800.0 PL=0
MOVL C00694 V=800.0 PL=0
MOVL C00695 V=800.0 PL=0
MOVL C00696 V=800.0 PL=0
MOVL C00697 V=800.0 PL=0
MOVL C00698 V=800.0 PL=0
MOVL C00699 V=800.0 PL=0
MOVL C00700 V=800.0 PL=0
MOVL C00701 V=800.0 PL=0
MOVL C00702 V=800.0 PL=0
MOVL C00703 V=800.0 PL=0
MOVL C00704 V=800.0 PL=0
MOVL C00705 V=800.0 PL=0
MOVL C00706 V=800.0 PL=0
MOVL C00707 V=800.0 PL=0
MOVL C00708 V=800.0 PL=0
MOVL C00709 V=800.0 PL=0
MOVL C00710 V=800.0 PL=0
MOVL C00711 V=800.0 PL=0
MOVL C00712 V=800.0 PL=0
MOVL C00713 V=800.0 PL=0
MOVL C00714 V=800.0 PL=0
MOVL C00715 V=800.0 PL=0
MOVL C00716 V=800.0 PL=0
MOVL C00717 V=800.0 PL=0
MOVL C00718 V=800.0 PL=0
MOVL C00719 V=800.0 PL=0
MOVL C00720 V=800.0 PL=0
MOVL C00721 V=800.0 PL=0
MOVL C00722 V=800.0 PL=0
MOVL C00723 V=800.0 PL=0
MOVL C00724 V=800.0 PL=0
MOVL C00725 V=800.0 PL=0
MOVL C00726 V=800.0 PL=0
MOVL C00727 V=800.0 PL=0
MOVL C00728 V=800.0 PL=0
MOVL C00729 V=800.0 PL=0
MOVL C00730 V=800.0 PL=0
MOVL C00731 V=800.0 PL=0
MOVL C00732 V=800.0 PL=0
MOVL C00733 V=800.0 PL=0
MOVL C00734 V=800.0 PL=0
MOVL C00735 V=800.0 PL=0
MOVL C00736 V=800.0 PL=0
MOVL C00737 V=800.0 PL=0
MOVL C00738 V=800.0 PL=0
MOVL C00739 V=800.0 PL=0
MOVL C00740 V=800.0 PL=0
MOVL C00741 V=800.0 PL=0
MOVL C00742 V=800.0 PL=0
MOVL C00743 V=800.0 PL=0
MOVL C00744 V=800.0 PL=0
MOVL C00745 V=800.0 PL=0
MOVL C00746 V=800.0 PL=0
MOVL C00747 V=800.0 PL=0
MOVL C00748 V=800.0 PL=0
MOVL C00749 V=800.0 PL=0
MOVL C00750 V=800.0 PL=0
MOVL C00751 V=800.0 PL=0
MOVL C00752 V=800.0 PL=0
MOVL C00753 V=800.0 PL=0
MOVL C00754 V=800.0 PL=0
MOVL C00755 V=800.0 PL=0
MOVL C00756 V=800.0 PL=0
MOVL C00757 V=800.0 PL=0
MOVL C00758 V=800.0 PL=0
MOVL C00759 V=800.0 PL=0
MOVL C00760 V=800.0 PL=0
MOVL C00761 V=800.0 PL=0
MOVL C00762 V=800.0 PL=0
MOVL C00763 V=800.0 PL=0
MOVL C00764 V=800.0 PL=0
MOVL C00765 V=800.0 PL=0
MOVL C00766 V=800.0 PL=0
MOVL C00767 V=800.0 PL=0
MOVL C00768 V=800.0 PL=0
MOVL C00769 V=800.0 PL=0
MOVL C00770 V=800.0 PL=0
MOVL C00771 V=800.0 PL=0
MOVL C00772 V=800.0 PL=0
MOVL C00773 V=800.0 PL=0
MOVL C00774 V=800.0 PL=0
MOVL C00775 V=800.0 PL=0
MOVL C00776 V=800.0 PL=0
MOVL C00777 V=800.0 PL=0
MOVL C00778 V=800.0 PL=0
MOVL C00779 V=800.0 PL=0
MOVL C00780 V=800.0 PL=0
MOVL C00781 V=800.0 PL=0
MOVL C00782 V=800.0 PL=0
MOVL C00783 V=800.0 PL=0
MOVL C00784 V=800.0 PL=0
MOVL C00785 V=800.0 PL=0
MOVL C00786 V=800.0 PL=0
MOVL C00787 V=800.0 PL=0
MOVL C00788 V=800.0 PL=0
MOVL C00789 V=800.0 PL=0
MOVL C00790 V=800.0 PL=0
'CALL JOB: TOOL OFF
MOVL C00791 V=800.0 PL=0
MOVJ C00792 VJ=25.00 PL=0
MOVL C00793 V=800.0 PL=0
'CALL JOB: TOOL ON
MOVL C00794 V=800.0 PL=0
MOVL C00795 V=800.0 PL=0
MOVL C00796 V=800.0 PL=0
MOVL C00797 V=800.0 PL=0
MOVL C00798 V=800.0 PL=0
MOVL C00799 V=800.0 PL=0
MOVL C00800 V=800.0 PL=0
MOVL C00801 V=800.0 PL=0
MOVL C00802 V=800.0 PL=0
MOVL C00803 V=800.0 PL=0
MOVL C00804 V=800.0 PL=0
MOVL C00805 V=800.0 PL=0
MOVL C00806 V=800.0 PL=0
MOVL C00807 V=800.0 PL=0
MOVL C00808 V=800.0 PL=0
MOVL C00809 V=800.0 PL=0
MOVL C00810 V=800.0 PL=0
MOVL C00811 V=800.0 PL=0
MOVL C00812 V=800.0 PL=0
MOVL C00813 V=800.0 PL=0
MOVL C00814 V=800.0 PL=0
MOVL C00815 V=800.0 PL=0
MOVL C00816 V=800.0 PL=0
MOVL C00817 V=800.0 PL=0
MOVL C00818 V=800.0 PL=0
MOVL C00819 V=800.0 PL=0
MOVL C00820 V=800.0 PL=0
MOVL C00821 V=800.0 PL=0
MOVL C00822 V=800.0 PL=0
MOVL C00823 V=800.0 PL=0
MOVL C00824 V=800.0 PL=0
MOVL C00825 V=800.0 PL=0
MOVL C00826 V=800.0 PL=0
MOVL C00827 V=800.0 PL=0
MOVL C00828 V=800.0 PL=0
MOVL C00829 V=800.0 PL=0
MOVL C00830 V=800.0 PL=0
MOVL C00831 V=800.0 PL=0
MOVL C00832 V=800.0 PL=0
MOVL C00833 V=800.0 PL=0
MOVL C00834 V=800.0 PL=0
MOVL C00835 V=800.0 PL=0
MOVL C00836 V=800.0 PL=0
MOVL C00837 V=800.0 PL=0
MOVL C00838 V=800.0 PL=0
MOVL C00839 V=800.0 PL=0
MOVL C00840 V=800.0 PL=0
MOVL C00841 V=800.0 PL=0
MOVL C00842 V=800.0 PL=0
MOVL C00843 V=800.0 PL=0
MOVL C00844 V=800.0 PL=0
MOVL C00845 V=800.0 PL=0
MOVL C00846 V=800.0 PL=0
MOVL C00847 V=800.0 PL=0
MOVL C00848 V=800.0 PL=0
MOVL C00849 V=800.0 PL=0
MOVL C00850 V=800.0 PL=0
MOVL C00851 V=800.0 PL=0
MOVL C00852 V=800.0 PL=0
MOVL C00853 V=800.0 PL=0
MOVL C00854 V=800.0 PL=0
MOVL C00855 V=800.0 PL=0
MOVL C00856 V=800.0 PL=0
MOVL C00857 V=800.0 PL=0
MOVL C00858 V=800.0 PL=0
MOVL C00859 V=800.0 PL=0
MOVL C00860 V=800.0 PL=0
MOVL C00861 V=800.0 PL=0
MOVL C00862 V=800.0 PL=0
MOVL C00863 V=800.0 PL=0
MOVL C00864 V=800.0 PL=0
MOVL C00865 V=800.0 PL=0
MOVL C00866 V=800.0 PL=0
MOVL C00867 V=800.0 PL=0
MOVL C00868 V=800.0 PL=0
MOVL C00869 V=800.0 PL=0
MOVL C00870 V=800.0 PL=0
MOVL C00871 V=800.0 PL=0
MOVL C00872 V=800.0 PL=0
MOVL C00873 V=800.0 PL=0
MOVL C00874 V=800.0 PL=0
'CALL JOB: TOOL OFF
MOVL C00875 V=800.0 PL=0
MOVJ C00876 VJ=25.00 PL=0
MOVL C00877 V=800.0 PL=0
'CALL JOB: TOOL ON
MOVL C00878 V=800.0 PL=0
MOVL C00879 V=800.0 PL=0
MOVL C00880 V=800.0 PL=0
MOVL C00881 V=800.0 PL=0
MOVL C00882 V=800.0 PL=0
MOVL C00883 V=800.0 PL=0
MOVL C00884 V=800.0 PL=0
MOVL C00885 V=800.0 PL=0
MOVL C00886 V=800.0 PL=0
MOVL C00887 V=800.0 PL=0
MOVL C00888 V=800.0 PL=0
MOVL C00889 V=800.0 PL=0
MOVL C00890 V=800.0 PL=0
MOVL C00891 V=800.0 PL=0
MOVL C00892 V=800.0 PL=0
MOVL C00893 V=800.0 PL=0
MOVL C00894 V=800.0 PL=0
MOVL C00895 V=800.0 PL=0
MOVL C00896 V=800.0 PL=0
MOVL C00897 V=800.0 PL=0
MOVL C00898 V=800.0 PL=0
MOVL C00899 V=800.0 PL=0
MOVL C00900 V=800.0 PL=0
MOVL C00901 V=800.0 PL=0
MOVL C00902 V=800.0 PL=0
MOVL C00903 V=800.0 PL=0
MOVL C00904 V=800.0 PL=0
MOVL C00905 V=800.0 PL=0
MOVL C00906 V=800.0 PL=0
MOVL C00907 V=800.0 PL=0
MOVL C00908 V=800.0 PL=0
MOVL C00909 V=800.0 PL=0
MOVL C00910 V=800.0 PL=0
MOVL C00911 V=800.0 PL=0
MOVL C00912 V=800.0 PL=0
MOVL C00913 V=800.0 PL=0
MOVL C00914 V=800.0 PL=0
MOVL C00915 V=800.0 PL=0
MOVL C00916 V=800.0 PL=0
MOVL C00917 V=800.0 PL=0
MOVL C00918 V=800.0 PL=0
MOVL C00919 V=800.0 PL=0
MOVL C00920 V=800.0 PL=0
MOVL C00921 V=800.0 PL=0
MOVL C00922 V=800.0 PL=0
MOVL C00923 V=800.0 PL=0
MOVL C00924 V=800.0 PL=0
MOVL C00925 V=800.0 PL=0
MOVL C00926 V=800.0 PL=0
MOVL C00927 V=800.0 PL=0
MOVL C00928 V=800.0 PL=0
MOVL C00929 V=800.0 PL=0
MOVL C00930 V=800.0 PL=0
MOVL C00931 V=800.0 PL=0
MOVL C00932 V=800.0 PL=0
MOVL C00933 V=800.0 PL=0
MOVL C00934 V=800.0 PL=0
MOVL C00935 V=800.0 PL=0
MOVL C00936 V=800.0 PL=0
MOVL C00937 V=800.0 PL=0
MOVL C00938 V=800.0 PL=0
MOVL C00939 V=800.0 PL=0
MOVL C00940 V=800.0 PL=0
MOVL C00941 V=800.0 PL=0
MOVL C00942 V=800.0 PL=0
MOVL C00943 V=800.0 PL=0
MOVL C00944 V=800.0 PL=0
MOVL C00945 V=800.0 PL=0
MOVL C00946 V=800.0 PL=0
MOVL C00947 V=800.0 PL=0
MOVL C00948 V=800.0 PL=0
MOVL C00949 V=800.0 PL=0
MOVL C00950 V=800.0 PL=0
MOVL C00951 V=800.0 PL=0
MOVL C00952 V=800.0 PL=0
MOVL C00953 V=800.0 PL=0
MOVL C00954 V=800.0 PL=0
MOVL C00955 V=800.0 PL=0
MOVL C00956 V=800.0 PL=0
MOVL C00957 V=800.0 PL=0
MOVL C00958 V=800.0 PL=0
MOVL C00959 V=800.0 PL=0
MOVL C00960 V=800.0 PL=0
MOVL C00961 V=800.0 PL=0
MOVL C00962 V=800.0 PL=0
MOVL C00963 V=800.0 PL=0
MOVL C00964 V=800.0 PL=0
MOVL C00965 V=800.0 PL=0
MOVL C00966 V=800.0 PL=0
MOVL C00967 V=800.0 PL=0
MOVL C00968 V=800.0 PL=0
MOVL C00969 V=800.0 PL=0
MOVL C00970 V=800.0 PL=0
MOVL C00971 V=800.0 PL=0
MOVL C00972 V=800.0 PL=0
MOVL C00973 V=800.0 PL=0
MOVL C00974 V=800.0 PL=0
MOVL C00975 V=800.0 PL=0
MOVL C00976 V=800.0 PL=0
MOVL C00977 V=800.0 PL=0
MOVL C00978 V=800.0 PL=0
MOVL C00979 V=800.0 PL=0
MOVL C00980 V=800.0 PL=0
MOVL C00981 V=800.0 PL=0
MOVL C00982 V=800.0 PL=0
MOVL C00983 V=800.0 PL=0
MOVL C00984 V=800.0 PL=0
MOVL C00985 V=800.0 PL=0
MOVL C00986 V=800.0 PL=0
MOVL C00987 V=800.0 PL=0
MOVL C00988 V=800.0 PL=0
MOVL C00989 V=800.0 PL=0
MOVL C00990 V=800.0 PL=0
MOVL C00991 V=800.0 PL=0
MOVL C00992 V=800.0 PL=0
MOVL C00993 V=800.0 PL=0
MOVL C00994 V=800.0 PL=0
MOVL C00995 V=800.0 PL=0
MOVL C00996 V=800.0 PL=0
MOVL C00997 V=800.0 PL=0
MOVL C00998 V=800.0 PL=0
MOVL C00999 V=800.0 PL=0
MOVL C01000 V=800.0 PL=0
MOVL C01001 V=800.0 PL=0
MOVL C01002 V=800.0 PL=0
MOVL C01003 V=800.0 PL=0
MOVL C01004 V=800.0 PL=0
MOVL C01005 V=800.0 PL=0
MOVL C01006 V=800.0 PL=0
MOVL C01007 V=800.0 PL=0
MOVL C01008 V=800.0 PL=0
MOVL C01009 V=800.0 PL=0
MOVL C01010 V=800.0 PL=0
MOVL C01011 V=800.0 PL=0
MOVL C01012 V=800.0 PL=0
MOVL C01013 V=800.0 PL=0
MOVL C01014 V=800.0 PL=0
MOVL C01015 V=800.0 PL=0
MOVL C01016 V=800.0 PL=0
MOVL C01017 V=800.0 PL=0
MOVL C01018 V=800.0 PL=0
MOVL C01019 V=800.0 PL=0
MOVL C01020 V=800.0 PL=0
MOVL C01021 V=800.0 PL=0
MOVL C01022 V=800.0 PL=0
MOVL C01023 V=800.0 PL=0
MOVL C01024 V=800.0 PL=0
MOVL C01025 V=800.0 PL=0
MOVL C01026 V=800.0 PL=0
MOVL C01027 V=800.0 PL=0
MOVL C01028 V=800.0 PL=0
MOVL C01029 V=800.0 PL=0
MOVL C01030 V=800.0 PL=0
MOVL C01031 V=800.0 PL=0
MOVL C01032 V=800.0 PL=0
MOVL C01033 V=800.0 PL=0
MOVL C01034 V=800.0 PL=0
MOVL C01035 V=800.0 PL=0
MOVL C01036 V=800.0 PL=0
MOVL C01037 V=800.0 PL=0
MOVL C01038 V=800.0 PL=0
MOVL C01039 V=800.0 PL=0
MOVL C01040 V=800.0 PL=0
MOVL C01041 V=800.0 PL=0
MOVL C01042 V=800.0 PL=0
MOVL C01043 V=800.0 PL=0
MOVL C01044 V=800.0 PL=0
MOVL C01045 V=800.0 PL=0
MOVL C01046 V=800.0 PL=0
MOVL C01047 V=800.0 PL=0
MOVL C01048 V=800.0 PL=0
MOVL C01049 V=800.0 PL=0
MOVL C01050 V=800.0 PL=0
MOVL C01051 V=800.0 PL=0
MOVL C01052 V=800.0 PL=0
MOVL C01053 V=800.0 PL=0
MOVL C01054 V=800.0 PL=0
MOVL C01055 V=800.0 PL=0
MOVL C01056 V=800.0 PL=0
MOVL C01057 V=800.0 PL=0
MOVL C01058 V=800.0 PL=0
MOVL C01059 V=800.0 PL=0
MOVL C01060 V=800.0 PL=0
MOVL C01061 V=800.0 PL=0
MOVL C01062 V=800.0 PL=0
MOVL C01063 V=800.0 PL=0
MOVL C01064 V=800.0 PL=0
MOVL C01065 V=800.0 PL=0
MOVL C01066 V=800.0 PL=0
MOVL C01067 V=800.0 PL=0
MOVL C01068 V=800.0 PL=0
MOVL C01069 V=800.0 PL=0
MOVL C01070 V=800.0 PL=0
MOVL C01071 V=800.0 PL=0
MOVL C01072 V=800.0 PL=0
MOVL C01073 V=800.0 PL=0
MOVL C01074 V=800.0 PL=0
MOVL C01075 V=800.0 PL=0
MOVL C01076 V=800.0 PL=0
MOVL C01077 V=800.0 PL=0
MOVL C01078 V=800.0 PL=0
MOVL C01079 V=800.0 PL=0
MOVL C01080 V=800.0 PL=0
MOVL C01081 V=800.0 PL=0
MOVL C01082 V=800.0 PL=0
MOVL C01083 V=800.0 PL=0
MOVL C01084 V=800.0 PL=0
MOVL C01085 V=800.0 PL=0
MOVL C01086 V=800.0 PL=0
MOVL C01087 V=800.0 PL=0
MOVL C01088 V=800.0 PL=0
MOVL C01089 V=800.0 PL=0
MOVL C01090 V=800.0 PL=0
MOVL C01091 V=800.0 PL=0
MOVL C01092 V=800.0 PL=0
MOVL C01093 V=800.0 PL=0
MOVL C01094 V=800.0 PL=0
MOVL C01095 V=800.0 PL=0
MOVL C01096 V=800.0 PL=0
MOVL C01097 V=800.0 PL=0
MOVL C01098 V=800.0 PL=0
MOVL C01099 V=800.0 PL=0
MOVL C01100 V=800.0 PL=0
MOVL C01101 V=800.0 PL=0
MOVL C01102 V=800.0 PL=0
MOVL C01103 V=800.0 PL=0
MOVL C01104 V=800.0 PL=0
MOVL C01105 V=800.0 PL=0
MOVL C01106 V=800.0 PL=0
MOVL C01107 V=800.0 PL=0
MOVL C01108 V=800.0 PL=0
MOVL C01109 V=800.0 PL=0
MOVL C01110 V=800.0 PL=0
MOVL C01111 V=800.0 PL=0
MOVL C01112 V=800.0 PL=0
MOVL C01113 V=800.0 PL=0
MOVL C01114 V=800.0 PL=0
MOVL C01115 V=800.0 PL=0
MOVL C01116 V=800.0 PL=0
MOVL C01117 V=800.0 PL=0
MOVL C01118 V=800.0 PL=0
MOVL C01119 V=800.0 PL=0
MOVL C01120 V=800.0 PL=0
MOVL C01121 V=800.0 PL=0
MOVL C01122 V=800.0 PL=0
MOVL C01123 V=800.0 PL=0
MOVL C01124 V=800.0 PL=0
MOVL C01125 V=800.0 PL=0
MOVL C01126 V=800.0 PL=0
MOVL C01127 V=800.0 PL=0
MOVL C01128 V=800.0 PL=0
MOVL C01129 V=800.0 PL=0
MOVL C01130 V=800.0 PL=0
MOVL C01131 V=800.0 PL=0
MOVL C01132 V=800.0 PL=0
MOVL C01133 V=800.0 PL=0
MOVL C01134 V=800.0 PL=0
MOVL C01135 V=800.0 PL=0
MOVL C01136 V=800.0 PL=0
MOVL C01137 V=800.0 PL=0
MOVL C01138 V=800.0 PL=0
MOVL C01139 V=800.0 PL=0
MOVL C01140 V=800.0 PL=0
MOVL C01141 V=800.0 PL=0
MOVL C01142 V=800.0 PL=0
MOVL C01143 V=800.0 PL=0
MOVL C01144 V=800.0 PL=0
MOVL C01145 V=800.0 PL=0
MOVL C01146 V=800.0 PL=0
MOVL C01147 V=800.0 PL=0
MOVL C01148 V=800.0 PL=0
MOVL C01149 V=800.0 PL=0
MOVL C01150 V=800.0 PL=0
MOVL C01151 V=800.0 PL=0
MOVL C01152 V=800.0 PL=0
MOVL C01153 V=800.0 PL=0
MOVL C01154 V=800.0 PL=0
MOVL C01155 V=800.0 PL=0
MOVL C01156 V=800.0 PL=0
MOVL C01157 V=800.0 PL=0
MOVL C01158 V=800.0 PL=0
MOVL C01159 V=800.0 PL=0
MOVL C01160 V=800.0 PL=0
MOVL C01161 V=800.0 PL=0
MOVL C01162 V=800.0 PL=0
MOVL C01163 V=800.0 PL=0
MOVL C01164 V=800.0 PL=0
MOVL C01165 V=800.0 PL=0
MOVL C01166 V=800.0 PL=0
MOVL C01167 V=800.0 PL=0
MOVL C01168 V=800.0 PL=0
MOVL C01169 V=800.0 PL=0
MOVL C01170 V=800.0 PL=0
MOVL C01171 V=800.0 PL=0
MOVL C01172 V=800.0 PL=0
MOVL C01173 V=800.0 PL=0
MOVL C01174 V=800.0 PL=0
MOVL C01175 V=800.0 PL=0
MOVL C01176 V=800.0 PL=0
MOVL C01177 V=800.0 PL=0
MOVL C01178 V=800.0 PL=0
MOVL C01179 V=800.0 PL=0
MOVL C01180 V=800.0 PL=0
MOVL C01181 V=800.0 PL=0
MOVL C01182 V=800.0 PL=0
MOVL C01183 V=800.0 PL=0
MOVL C01184 V=800.0 PL=0
MOVL C01185 V=800.0 PL=0
MOVL C01186 V=800.0 PL=0
MOVL C01187 V=800.0 PL=0
MOVL C01188 V=800.0 PL=0
MOVL C01189 V=800.0 PL=0
MOVL C01190 V=800.0 PL=0
MOVL C01191 V=800.0 PL=0
MOVL C01192 V=800.0 PL=0
MOVL C01193 V=800.0 PL=0
MOVL C01194 V=800.0 PL=0
MOVL C01195 V=800.0 PL=0
MOVL C01196 V=800.0 PL=0
MOVL C01197 V=800.0 PL=0
MOVL C01198 V=800.0 PL=0
MOVL C01199 V=800.0 PL=0
MOVL C01200 V=800.0 PL=0
MOVL C01201 V=800.0 PL=0
MOVL C01202 V=800.0 PL=0
MOVL C01203 V=800.0 PL=0
MOVL C01204 V=800.0 PL=0
MOVL C01205 V=800.0 PL=0
MOVL C01206 V=800.0 PL=0
MOVL C01207 V=800.0 PL=0
MOVL C01208 V=800.0 PL=0
MOVL C01209 V=800.0 PL=0
MOVL C01210 V=800.0 PL=0
MOVL C01211 V=800.0 PL=0
MOVL C01212 V=800.0 PL=0
MOVL C01213 V=800.0 PL=0
MOVL C01214 V=800.0 PL=0
MOVL C01215 V=800.0 PL=0
MOVL C01216 V=800.0 PL=0
MOVL C01217 V=800.0 PL=0
MOVL C01218 V=800.0 PL=0
MOVL C01219 V=800.0 PL=0
MOVL C01220 V=800.0 PL=0
MOVL C01221 V=800.0 PL=0
MOVL C01222 V=800.0 PL=0
MOVL C01223 V=800.0 PL=0
MOVL C01224 V=800.0 PL=0
MOVL C01225 V=800.0 PL=0
MOVL C01226 V=800.0 PL=0
MOVL C01227 V=800.0 PL=0
MOVL C01228 V=800.0 PL=0
MOVL C01229 V=800.0 PL=0
MOVL C01230 V=800.0 PL=0
MOVL C01231 V=800.0 PL=0
MOVL C01232 V=800.0 PL=0
MOVL C01233 V=800.0 PL=0
MOVL C01234 V=800.0 PL=0
MOVL C01235 V=800.0 PL=0
MOVL C01236 V=800.0 PL=0
MOVL C01237 V=800.0 PL=0
MOVL C01238 V=800.0 PL=0
MOVL C01239 V=800.0 PL=0
MOVL C01240 V=800.0 PL=0
MOVL C01241 V=800.0 PL=0
MOVL C01242 V=800.0 PL=0
MOVL C01243 V=800.0 PL=0
MOVL C01244 V=800.0 PL=0
MOVL C01245 V=800.0 PL=0
MOVL C01246 V=800.0 PL=0
MOVL C01247 V=800.0 PL=0
MOVL C01248 V=800.0 PL=0
MOVL C01249 V=800.0 PL=0
MOVL C01250 V=800.0 PL=0
MOVL C01251 V=800.0 PL=0
MOVL C01252 V=800.0 PL=0
MOVL C01253 V=800.0 PL=0
MOVL C01254 V=800.0 PL=0
MOVL C01255 V=800.0 PL=0
MOVL C01256 V=800.0 PL=0
MOVL C01257 V=800.0 PL=0
MOVL C01258 V=800.0 PL=0
MOVL C01259 V=800.0 PL=0
MOVL C01260 V=800.0 PL=0
MOVL C01261 V=800.0 PL=0
MOVL C01262 V=800.0 PL=0
MOVL C01263 V=800.0 PL=0
MOVL C01264 V=800.0 PL=0
MOVL C01265 V=800.0 PL=0
MOVL C01266 V=800.0 PL=0
MOVL C01267 V=800.0 PL=0
MOVL C01268 V=800.0 PL=0
MOVL C01269 V=800.0 PL=0
MOVL C01270 V=800.0 PL=0
MOVL C01271 V=800.0 PL=0
MOVL C01272 V=800.0 PL=0
MOVL C01273 V=800.0 PL=0
MOVL C01274 V=800.0 PL=0
MOVL C01275 V=800.0 PL=0
MOVL C01276 V=800.0 PL=0
MOVL C01277 V=800.0 PL=0
MOVL C01278 V=800.0 PL=0
MOVL C01279 V=800.0 PL=0
MOVL C01280 V=800.0 PL=0
MOVL C01281 V=800.0 PL=0
MOVL C01282 V=800.0 PL=0
MOVL C01283 V=800.0 PL=0
MOVL C01284 V=800.0 PL=0
MOVL C01285 V=800.0 PL=0
MOVL C01286 V=800.0 PL=0
MOVL C01287 V=800.0 PL=0
MOVL C01288 V=800.0 PL=0
MOVL C01289 V=800.0 PL=0
MOVL C01290 V=800.0 PL=0
MOVL C01291 V=800.0 PL=0
MOVL C01292 V=800.0 PL=0
MOVL C01293 V=800.0 PL=0
MOVL C01294 V=800.0 PL=0
MOVL C01295 V=800.0 PL=0
MOVL C01296 V=800.0 PL=0
MOVL C01297 V=800.0 PL=0
MOVL C01298 V=800.0 PL=0
MOVL C01299 V=800.0 PL=0
MOVL C01300 V=800.0 PL=0
MOVL C01301 V=800.0 PL=0
MOVL C01302 V=800.0 PL=0
MOVL C01303 V=800.0 PL=0
MOVL C01304 V=800.0 PL=0
MOVL C01305 V=800.0 PL=0
MOVL C01306 V=800.0 PL=0
MOVL C01307 V=800.0 PL=0
MOVL C01308 V=800.0 PL=0
MOVL C01309 V=800.0 PL=0
MOVL C01310 V=800.0 PL=0
MOVL C01311 V=800.0 PL=0
MOVL C01312 V=800.0 PL=0
MOVL C01313 V=800.0 PL=0
MOVL C01314 V=800.0 PL=0
MOVL C01315 V=800.0 PL=0
MOVL C01316 V=800.0 PL=0
MOVL C01317 V=800.0 PL=0
MOVL C01318 V=800.0 PL=0
MOVL C01319 V=800.0 PL=0
MOVL C01320 V=800.0 PL=0
MOVL C01321 V=800.0 PL=0
MOVL C01322 V=800.0 PL=0
MOVL C01323 V=800.0 PL=0
MOVL C01324 V=800.0 PL=0
MOVL C01325 V=800.0 PL=0
MOVL C01326 V=800.0 PL=0
MOVL C01327 V=800.0 PL=0
MOVL C01328 V=800.0 PL=0
MOVL C01329 V=800.0 PL=0
MOVL C01330 V=800.0 PL=0
MOVL C01331 V=800.0 PL=0
MOVL C01332 V=800.0 PL=0
MOVL C01333 V=800.0 PL=0
MOVL C01334 V=800.0 PL=0
MOVL C01335 V=800.0 PL=0
MOVL C01336 V=800.0 PL=0
MOVL C01337 V=800.0 PL=0
MOVL C01338 V=800.0 PL=0
MOVL C01339 V=800.0 PL=0
MOVL C01340 V=800.0 PL=0
MOVL C01341 V=800.0 PL=0
MOVL C01342 V=800.0 PL=0
MOVL C01343 V=800.0 PL=0
MOVL C01344 V=800.0 PL=0
MOVL C01345 V=800.0 PL=0
MOVL C01346 V=800.0 PL=0
MOVL C01347 V=800.0 PL=0
MOVL C01348 V=800.0 PL=0
MOVL C01349 V=800.0 PL=0
MOVL C01350 V=800.0 PL=0
MOVL C01351 V=800.0 PL=0
MOVL C01352 V=800.0 PL=0
MOVL C01353 V=800.0 PL=0
MOVL C01354 V=800.0 PL=0
MOVL C01355 V=800.0 PL=0
MOVL C01356 V=800.0 PL=0
MOVL C01357 V=800.0 PL=0
MOVL C01358 V=800.0 PL=0
MOVL C01359 V=800.0 PL=0
MOVL C01360 V=800.0 PL=0
MOVL C01361 V=800.0 PL=0
MOVL C01362 V=800.0 PL=0
MOVL C01363 V=800.0 PL=0
MOVL C01364 V=800.0 PL=0
MOVL C01365 V=800.0 PL=0
MOVL C01366 V=800.0 PL=0
MOVL C01367 V=800.0 PL=0
MOVL C01368 V=800.0 PL=0
MOVL C01369 V=800.0 PL=0
MOVL C01370 V=800.0 PL=0
MOVL C01371 V=800.0 PL=0
MOVL C01372 V=800.0 PL=0
MOVL C01373 V=800.0 PL=0
MOVL C01374 V=800.0 PL=0
MOVL C01375 V=800.0 PL=0
MOVL C01376 V=800.0 PL=0
MOVL C01377 V=800.0 PL=0
MOVL C01378 V=800.0 PL=0
MOVL C01379 V=800.0 PL=0
MOVL C01380 V=800.0 PL=0
MOVL C01381 V=800.0 PL=0
MOVL C01382 V=800.0 PL=0
MOVL C01383 V=800.0 PL=0
MOVL C01384 V=800.0 PL=0
MOVL C01385 V=800.0 PL=0
MOVL C01386 V=800.0 PL=0
MOVL C01387 V=800.0 PL=0
MOVL C01388 V=800.0 PL=0
MOVL C01389 V=800.0 PL=0
MOVL C01390 V=800.0 PL=0
MOVL C01391 V=800.0 PL=0
MOVL C01392 V=800.0 PL=0
MOVL C01393 V=800.0 PL=0
MOVL C01394 V=800.0 PL=0
MOVL C01395 V=800.0 PL=0
MOVL C01396 V=800.0 PL=0
MOVL C01397 V=800.0 PL=0
MOVL C01398 V=800.0 PL=0
MOVL C01399 V=800.0 PL=0
MOVL C01400 V=800.0 PL=0
MOVL C01401 V=800.0 PL=0
MOVL C01402 V=800.0 PL=0
MOVL C01403 V=800.0 PL=0
MOVL C01404 V=800.0 PL=0
MOVL C01405 V=800.0 PL=0
MOVL C01406 V=800.0 PL=0
MOVL C01407 V=800.0 PL=0
MOVL C01408 V=800.0 PL=0
MOVL C01409 V=800.0 PL=0
MOVL C01410 V=800.0 PL=0
MOVL C01411 V=800.0 PL=0
MOVL C01412 V=800.0 PL=0
MOVL C01413 V=800.0 PL=0
MOVL C01414 V=800.0 PL=0
MOVL C01415 V=800.0 PL=0
MOVL C01416 V=800.0 PL=0
MOVL C01417 V=800.0 PL=0
MOVL C01418 V=800.0 PL=0
MOVL C01419 V=800.0 PL=0
MOVL C01420 V=800.0 PL=0
MOVL C01421 V=800.0 PL=0
MOVL C01422 V=800.0 PL=0
MOVL C01423 V=800.0 PL=0
MOVL C01424 V=800.0 PL=0
MOVL C01425 V=800.0 PL=0
MOVL C01426 V=800.0 PL=0
MOVL C01427 V=800.0 PL=0
MOVL C01428 V=800.0 PL=0
MOVL C01429 V=800.0 PL=0
MOVL C01430 V=800.0 PL=0
MOVL C01431 V=800.0 PL=0
MOVL C01432 V=800.0 PL=0
MOVL C01433 V=800.0 PL=0
MOVL C01434 V=800.0 PL=0
MOVL C01435 V=800.0 PL=0
MOVL C01436 V=800.0 PL=0
MOVL C01437 V=800.0 PL=0
MOVL C01438 V=800.0 PL=0
MOVL C01439 V=800.0 PL=0
MOVL C01440 V=800.0 PL=0
MOVL C01441 V=800.0 PL=0
MOVL C01442 V=800.0 PL=0
MOVL C01443 V=800.0 PL=0
MOVL C01444 V=800.0 PL=0
MOVL C01445 V=800.0 PL=0
MOVL C01446 V=800.0 PL=0
MOVL C01447 V=800.0 PL=0
MOVL C01448 V=800.0 PL=0
MOVL C01449 V=800.0 PL=0
MOVL C01450 V=800.0 PL=0
MOVL C01451 V=800.0 PL=0
MOVL C01452 V=800.0 PL=0
MOVL C01453 V=800.0 PL=0
MOVL C01454 V=800.0 PL=0
MOVL C01455 V=800.0 PL=0
MOVL C01456 V=800.0 PL=0
MOVL C01457 V=800.0 PL=0
MOVL C01458 V=800.0 PL=0
MOVL C01459 V=800.0 PL=0
MOVL C01460 V=800.0 PL=0
MOVL C01461 V=800.0 PL=0
MOVL C01462 V=800.0 PL=0
MOVL C01463 V=800.0 PL=0
MOVL C01464 V=800.0 PL=0
MOVL C01465 V=800.0 PL=0
MOVL C01466 V=800.0 PL=0
MOVL C01467 V=800.0 PL=0
MOVL C01468 V=800.0 PL=0
MOVL C01469 V=800.0 PL=0
MOVL C01470 V=800.0 PL=0
MOVL C01471 V=800.0 PL=0
MOVL C01472 V=800.0 PL=0
MOVL C01473 V=800.0 PL=0
MOVL C01474 V=800.0 PL=0
MOVL C01475 V=800.0 PL=0
MOVL C01476 V=800.0 PL=0
MOVL C01477 V=800.0 PL=0
MOVL C01478 V=800.0 PL=0
MOVL C01479 V=800.0 PL=0
MOVL C01480 V=800.0 PL=0
MOVL C01481 V=800.0 PL=0
MOVL C01482 V=800.0 PL=0
MOVL C01483 V=800.0 PL=0
MOVL C01484 V=800.0 PL=0
MOVL C01485 V=800.0 PL=0
MOVL C01486 V=800.0 PL=0
MOVL C01487 V=800.0 PL=0
MOVL C01488 V=800.0 PL=0
MOVL C01489 V=800.0 PL=0
MOVL C01490 V=800.0 PL=0
MOVL C01491 V=800.0 PL=0
MOVL C01492 V=800.0 PL=0
MOVL C01493 V=800.0 PL=0
MOVL C01494 V=800.0 PL=0
MOVL C01495 V=800.0 PL=0
MOVL C01496 V=800.0 PL=0
MOVL C01497 V=800.0 PL=0
MOVL C01498 V=800.0 PL=0
MOVL C01499 V=800.0 PL=0
MOVL C01500 V=800.0 PL=0
MOVL C01501 V=800.0 PL=0
MOVL C01502 V=800.0 PL=0
MOVL C01503 V=800.0 PL=0
MOVL C01504 V=800.0 PL=0
MOVL C01505 V=800.0 PL=0
MOVL C01506 V=800.0 PL=0
MOVL C01507 V=800.0 PL=0
MOVL C01508 V=800.0 PL=0
MOVL C01509 V=800.0 PL=0
MOVL C01510 V=800.0 PL=0
MOVL C01511 V=800.0 PL=0
MOVL C01512 V=800.0 PL=0
MOVL C01513 V=800.0 PL=0
MOVL C01514 V=800.0 PL=0
MOVL C01515 V=800.0 PL=0
MOVL C01516 V=800.0 PL=0
MOVL C01517 V=800.0 PL=0
MOVL C01518 V=800.0 PL=0
MOVL C01519 V=800.0 PL=0
MOVL C01520 V=800.0 PL=0
MOVL C01521 V=800.0 PL=0
MOVL C01522 V=800.0 PL=0
MOVL C01523 V=800.0 PL=0
MOVL C01524 V=800.0 PL=0
MOVL C01525 V=800.0 PL=0
MOVL C01526 V=800.0 PL=0
MOVL C01527 V=800.0 PL=0
MOVL C01528 V=800.0 PL=0
MOVL C01529 V=800.0 PL=0
MOVL C01530 V=800.0 PL=0
MOVL C01531 V=800.0 PL=0
MOVL C01532 V=800.0 PL=0
MOVL C01533 V=800.0 PL=0
MOVL C01534 V=800.0 PL=0
MOVL C01535 V=800.0 PL=0
MOVL C01536 V=800.0 PL=0
MOVL C01537 V=800.0 PL=0
MOVL C01538 V=800.0 PL=0
MOVL C01539 V=800.0 PL=0
MOVL C01540 V=800.0 PL=0
MOVL C01541 V=800.0 PL=0
MOVL C01542 V=800.0 PL=0
MOVL C01543 V=800.0 PL=0
MOVL C01544 V=800.0 PL=0
MOVL C01545 V=800.0 PL=0
MOVL C01546 V=800.0 PL=0
MOVL C01547 V=800.0 PL=0
MOVL C01548 V=800.0 PL=0
MOVL C01549 V=800.0 PL=0
MOVL C01550 V=800.0 PL=0
MOVL C01551 V=800.0 PL=0
MOVL C01552 V=800.0 PL=0
MOVL C01553 V=800.0 PL=0
MOVL C01554 V=800.0 PL=0
MOVL C01555 V=800.0 PL=0
MOVL C01556 V=800.0 PL=0
MOVL C01557 V=800.0 PL=0
MOVL C01558 V=800.0 PL=0
MOVL C01559 V=800.0 PL=0
MOVL C01560 V=800.0 PL=0
MOVL C01561 V=800.0 PL=0
MOVL C01562 V=800.0 PL=0
MOVL C01563 V=800.0 PL=0
MOVL C01564 V=800.0 PL=0
MOVL C01565 V=800.0 PL=0
MOVL C01566 V=800.0 PL=0
MOVL C01567 V=800.0 PL=0
MOVL C01568 V=800.0 PL=0
MOVL C01569 V=800.0 PL=0
MOVL C01570 V=800.0 PL=0
MOVL C01571 V=800.0 PL=0
MOVL C01572 V=800.0 PL=0
MOVL C01573 V=800.0 PL=0
MOVL C01574 V=800.0 PL=0
MOVL C01575 V=800.0 PL=0
MOVL C01576 V=800.0 PL=0
MOVL C01577 V=800.0 PL=0
MOVL C01578 V=800.0 PL=0
MOVL C01579 V=800.0 PL=0
MOVL C01580 V=800.0 PL=0
MOVL C01581 V=800.0 PL=0
MOVL C01582 V=800.0 PL=0
MOVL C01583 V=800.0 PL=0
MOVL C01584 V=800.0 PL=0
MOVL C01585 V=800.0 PL=0
MOVL C01586 V=800.0 PL=0
MOVL C01587 V=800.0 PL=0
MOVL C01588 V=800.0 PL=0
MOVL C01589 V=800.0 PL=0
MOVL C01590 V=800.0 PL=0
MOVL C01591 V=800.0 PL=0
MOVL C01592 V=800.0 PL=0
MOVL C01593 V=800.0 PL=0
MOVL C01594 V=800.0 PL=0
MOVL C01595 V=800.0 PL=0
MOVL C01596 V=800.0 PL=0
MOVL C01597 V=800.0 PL=0
MOVL C01598 V=800.0 PL=0
MOVL C01599 V=800.0 PL=0
MOVL C01600 V=800.0 PL=0
MOVL C01601 V=800.0 PL=0
MOVL C01602 V=800.0 PL=0
MOVL C01603 V=800.0 PL=0
MOVL C01604 V=800.0 PL=0
MOVL C01605 V=800.0 PL=0
MOVL C01606 V=800.0 PL=0
MOVL C01607 V=800.0 PL=0
MOVL C01608 V=800.0 PL=0
MOVL C01609 V=800.0 PL=0
MOVL C01610 V=800.0 PL=0
MOVL C01611 V=800.0 PL=0
MOVL C01612 V=800.0 PL=0
MOVL C01613 V=800.0 PL=0
MOVL C01614 V=800.0 PL=0
MOVL C01615 V=800.0 PL=0
MOVL C01616 V=800.0 PL=0
MOVL C01617 V=800.0 PL=0
MOVL C01618 V=800.0 PL=0
MOVL C01619 V=800.0 PL=0
MOVL C01620 V=800.0 PL=0
